LIN {X 0,Y 462.076,Z 805.62,A -85,B 0,C 180,E1 21191.71,E2 21191.71} C_VEL
LIN {X 0,Y 459.334,Z 826.839,A -85,B 0,C 180,E1 21190.527,E2 21190.527} C_VEL
LIN {X 0,Y 456.263,Z 847.373,A -85,B 0,C 180,E1 21189.127,E2 21189.127} C_VEL
LIN {X 0,Y 453.108,Z 867.434,A -85,B 0,C 180,E1 21187.515,E2 21187.515} C_VEL
LIN {X 0,Y 449.988,Z 885.995,A -85,B 0,C 180,E1 21185.755,E2 21185.755} C_VEL
LIN {X 0,Y 446.558,Z 905.771,A -85,B 0,C 180,E1 21183.572,E2 21183.572} C_VEL
LIN {X 0,Y 443.731,Z 922.212,A -85,B 0,C 180,E1 21181.463,E2 21181.463} C_VEL
LIN {X 0,Y 440.914,Z 938.619,A -85,B 0,C 180,E1 21179.028,E2 21179.028} C_VEL
LIN {X 0,Y 438.594,Z 953.242,A -85,B 0,C 180,E1 21176.537,E2 21176.537} C_VEL
LIN {X 0,Y 436.587,Z 966.429,A -85,B 0,C 180,E1 21173.911,E2 21173.911} C_VEL
LIN {X 0,Y 434.952,Z 978.265,A -85,B 0,C 180,E1 21171.154,E2 21171.154} C_VEL
LIN {X 0,Y 433.708,Z 988.605,A -85,B 0,C 180,E1 21168.27,E2 21168.27} C_VEL
LIN {X 0,Y 432.814,Z 997.995,A -85,B 0,C 180,E1 21165.131,E2 21165.131} C_VEL
LIN {X 0,Y 432.337,Z 1004.562,A -85,B 0,C 180,E1 21162.419,E2 21162.419} C_VEL
LIN {X 0,Y 432.051,Z 1010.43,A -85,B 0,C 180,E1 21159.322,E2 21159.322} C_VEL
LIN {X 0,Y 431.943,Z 1014.119,A -85,B 0,C 180,E1 21156.646,E2 21156.646} C_VEL
LIN {X 0,Y 431.896,Z 1016.848,A -85,B 0,C 180,E1 21153.584,E2 21153.584} C_VEL
LIN {X 0,Y 431.89,Z 1017.848,A -85,B 0,C 180,E1 21150.929,E2 21150.929} C_VEL
LIN {X 0,Y 431.907,Z 1017.69,A -85,B 0,C 180,E1 21148.143,E2 21148.143} C_VEL
LIN {X 0,Y 431.91,Z 1015.955,A -85,B 0,C 180,E1 21145.22,E2 21145.22} C_VEL
LIN {X 0,Y 431.948,Z 1013.161,A -85,B 0,C 180,E1 21142.553,E2 21142.553} C_VEL
LIN {X 0,Y 432.128,Z 1008.339,A -85,B 0,C 180,E1 21139.469,E2 21139.469} C_VEL
LIN {X 0,Y 432.462,Z 1002.684,A -85,B 0,C 180,E1 21136.743,E2 21136.743} C_VEL
LIN {X 0,Y 433.106,Z 994.557,A -85,B 0,C 180,E1 21133.644,E2 21133.644} C_VEL
LIN {X 0,Y 434.06,Z 985.527,A -85,B 0,C 180,E1 21130.809,E2 21130.809} C_VEL
LIN {X 0,Y 435.394,Z 974.873,A -85,B 0,C 180,E1 21128.021,E2 21128.021} C_VEL
LIN {X 0,Y 436.966,Z 963.844,A -85,B 0,C 180,E1 21125.537,E2 21125.537} C_VEL
LIN {X 0,Y 439.061,Z 950.109,A -85,B 0,C 180,E1 21122.91,E2 21122.91} C_VEL
LIN {X 0,Y 441.553,Z 935.071,A -85,B 0,C 180,E1 21120.404,E2 21120.404} C_VEL
LIN {X 0,Y 444.365,Z 918.393,A -85,B 0,C 180,E1 21118.024,E2 21118.024} C_VEL
LIN {X 0,Y 447.495,Z 900.571,A -85,B 0,C 180,E1 21115.815,E2 21115.815} C_VEL
LIN {X 0,Y 450.434,Z 883.294,A -85,B 0,C 180,E1 21113.973,E2 21113.973} C_VEL
LIN {X 0,Y 453.737,Z 863.496,A -85,B 0,C 180,E1 21112.148,E2 21112.148} C_VEL
LIN {X 0,Y 456.694,Z 844.645,A -85,B 0,C 180,E1 21110.674,E2 21110.674} C_VEL
LIN {X 0,Y 459.9,Z 822.472,A -85,B 0,C 180,E1 21109.215,E2 21109.215} C_VEL
LIN {X 0,Y 462.377,Z 803.115,A -85,B 0,C 180,E1 21108.162,E2 21108.162} C_VEL
LIN {X 0,Y 465.009,Z 779.05,A -85,B 0,C 180,E1 21107.112,E2 21107.112} C_VEL
LIN {X 0,Y 467.004,Z 756.997,A -85,B 0,C 180,E1 21106.38,E2 21106.38} C_VEL
LIN {X 0,Y 468.458,Z 733.73,A -85,B 0,C 180,E1 21105.834,E2 21105.834} C_VEL
LIN {X 0,Y 474.656,Z 531.518,A -85,B 0,C 180,E1 21102.256,E2 21102.256} C_VEL
LIN {X 0,Y 477.415,Z 442.989,A -85,B 0,C 180,E1 21100.663,E2 21100.663} C_VEL
LIN {X 0,Y 466.316,Z 425.345,A -85,B 0,C 180,E1 21098.644,E2 21098.644} C_VEL
LIN {X 0,Y 456.213,Z 410.687,A -85,B 0,C 180,E1 21096.671,E2 21096.671} C_VEL
LIN {X 0,Y 446.549,Z 397.276,A -85,B 0,C 180,E1 21094.622,E2 21094.622} C_VEL
LIN {X 0,Y 442.193,Z 391.483,A -85,B 0,C 180,E1 21093.64,E2 21093.64} C_VEL
LIN {X 0,Y 438.295,Z 386.486,A -85,B 0,C 180,E1 21092.728,E2 21092.728} C_VEL
LIN {X 0,Y 436.603,Z 384.125,A -85,B 0,C 180,E1 21092.248,E2 21092.248} C_VEL
LIN {X 0,Y 435.545,Z 381.762,A -85,B 0,C 180,E1 21091.715,E2 21091.715} C_VEL
LIN {X 0,Y 433.675,Z 378.949,A -85,B 0,C 180,E1 21090.939,E2 21090.939} C_VEL
LIN {X 0,Y 433.213,Z 377.052,A -85,B 0,C 180,E1 21090.514,E2 21090.514} C_VEL
LIN {X 0,Y 433.202,Z 377.083,A -85,B 0,C 180,E1 21086.748,E2 21086.748} C_VEL
LIN {X 0,Y 433.196,Z 377.04,A -85,B 0,C 180,E1 21082.954,E2 21082.954} C_VEL
LIN {X 0,Y 433.235,Z 377.058,A -85,B 0,C 180,E1 21079.41,E2 21079.41} C_VEL
LIN {X 0,Y 433.241,Z 377.062,A -85,B 0,C 180,E1 21075.528,E2 21075.528} C_VEL
LIN {X 0,Y 433.199,Z 377.077,A -85,B 0,C 180,E1 21071.854,E2 21071.854} C_VEL
LIN {X 0,Y 433.177,Z 377.084,A -85,B 0,C 180,E1 21068.227,E2 21068.227} C_VEL
LIN {X 0,Y 433.183,Z 377.087,A -85,B 0,C 180,E1 21064.434,E2 21064.434} C_VEL
LIN {X 0,Y 433.218,Z 377.081,A -85,B 0,C 180,E1 21060.793,E2 21060.793} C_VEL
LIN {X 0,Y 433.232,Z 377.079,A -85,B 0,C 180,E1 21057.089,E2 21057.089} C_VEL
LIN {X 0,Y 433.208,Z 377.083,A -85,B 0,C 180,E1 21053.373,E2 21053.373} C_VEL
LIN {X 0,Y 433.195,Z 377.086,A -85,B 0,C 180,E1 21049.763,E2 21049.763} C_VEL
LIN {X 0,Y 433.206,Z 377.086,A -85,B 0,C 180,E1 21045.975,E2 21045.975} C_VEL
LIN {X 0,Y 433.24,Z 377.03,A -85,B 0,C 180,E1 21042.37,E2 21042.37} C_VEL
LIN {X 0,Y 433.253,Z 377.074,A -85,B 0,C 180,E1 21038.615,E2 21038.615} C_VEL
LIN {X 0,Y 433.225,Z 377.048,A -85,B 0,C 180,E1 21034.871,E2 21034.871} C_VEL
LIN {X 0,Y 433.213,Z 377.045,A -85,B 0,C 180,E1 21031.159,E2 21031.159} C_VEL
LIN {X 0,Y 433.277,Z 377.224,A -85,B 0,C 180,E1 21028.021,E2 21028.021} C_VEL
LIN {X 0,Y 434.29,Z 380.161,A -85,B 0,C 180,E1 21027.715,E2 21027.715} C_VEL
LIN {X 0,Y 436.695,Z 382.725,A -85,B 0,C 180,E1 21027.137,E2 21027.137} C_VEL
LIN {X 0,Y 438.075,Z 383.765,A -85,B 0,C 180,E1 21026.824,E2 21026.824} C_VEL
LIN {X 0,Y 440.43,Z 387.482,A -85,B 0,C 180,E1 21026.246,E2 21026.246} C_VEL
LIN {X 0,Y 442.869,Z 389.914,A -85,B 0,C 180,E1 21025.702,E2 21025.702} C_VEL
LIN {X 0,Y 446.063,Z 394.129,A -85,B 0,C 180,E1 21024.982,E2 21024.982} C_VEL
LIN {X 0,Y 447.593,Z 395.982,A -85,B 0,C 180,E1 21024.65,E2 21024.65} C_VEL
LIN {X 0,Y 456.054,Z 406.862,A -85,B 0,C 180,E1 21022.882,E2 21022.882} C_VEL
LIN {X 0,Y 467.056,Z 421.727,A -85,B 0,C 180,E1 21020.758,E2 21020.758} C_VEL
LIN {X 0,Y 477.318,Z 436.615,A -85,B 0,C 180,E1 21018.921,E2 21018.921} C_VEL
LIN {X 0,Y 470.969,Z 637.153,A -85,B 0,C 180,E1 21015.357,E2 21015.357} C_VEL
LIN {X 0,Y 469.061,Z 701.067,A -85,B 0,C 180,E1 21014.235,E2 21014.235} C_VEL
LIN {X 0,Y 467.994,Z 708.752,A -85,B 0,C 180,E1 21014.173,E2 21014.173} C_VEL
LIN {X 0,Y 462.507,Z 728.147,A -85,B 0,C 180,E1 21014.247,E2 21014.247} C_VEL
LIN {X 0,Y 461.232,Z 735.659,A -85,B 0,C 180,E1 21014.106,E2 21014.106} C_VEL
LIN {X 0,Y 459.247,Z 757.338,A -85,B 0,C 180,E1 21013.336,E2 21013.336} C_VEL
LIN {X 0,Y 456.812,Z 778.149,A -85,B 0,C 180,E1 21012.381,E2 21012.381} C_VEL
LIN {X 0,Y 454.246,Z 797.149,A -85,B 0,C 180,E1 21011.32,E2 21011.32} C_VEL
LIN {X 0,Y 450.876,Z 818.833,A -85,B 0,C 180,E1 21009.852,E2 21009.852} C_VEL
LIN {X 0,Y 447.624,Z 838.068,A -85,B 0,C 180,E1 21008.3,E2 21008.3} C_VEL
LIN {X 0,Y 444.229,Z 856.539,A -85,B 0,C 180,E1 21006.532,E2 21006.532} C_VEL
LIN {X 0,Y 440.833,Z 874.551,A -85,B 0,C 180,E1 21004.538,E2 21004.538} C_VEL
LIN {X 0,Y 437.468,Z 891.506,A -85,B 0,C 180,E1 21002.327,E2 21002.327} C_VEL
LIN {X 0,Y 434.438,Z 907.273,A -85,B 0,C 180,E1 20999.958,E2 20999.958} C_VEL
LIN {X 0,Y 431.785,Z 921.227,A -85,B 0,C 180,E1 20997.515,E2 20997.515} C_VEL
LIN {X 0,Y 429.286,Z 935.376,A -85,B 0,C 180,E1 20994.636,E2 20994.636} C_VEL
LIN {X 0,Y 427.507,Z 946.566,A -85,B 0,C 180,E1 20991.972,E2 20991.972} C_VEL
LIN {X 0,Y 425.948,Z 958.005,A -85,B 0,C 180,E1 20988.756,E2 20988.756} C_VEL
LIN {X 0,Y 425.016,Z 966.889,A -85,B 0,C 180,E1 20985.807,E2 20985.807} C_VEL
LIN {X 0,Y 424.426,Z 973.858,A -85,B 0,C 180,E1 20982.93,E2 20982.93} C_VEL
LIN {X 0,Y 424.076,Z 979.744,A -85,B 0,C 180,E1 20979.909,E2 20979.909} C_VEL
LIN {X 0,Y 423.936,Z 983.747,A -85,B 0,C 180,E1 20977.043,E2 20977.043} C_VEL
LIN {X 0,Y 423.913,Z 986.485,A -85,B 0,C 180,E1 20974.192,E2 20974.192} C_VEL
LIN {X 0,Y 423.905,Z 987.795,A -85,B 0,C 180,E1 20971.216,E2 20971.216} C_VEL
LIN {X 0,Y 423.909,Z 987.765,A -85,B 0,C 180,E1 20968.513,E2 20968.513} C_VEL
LIN {X 0,Y 423.907,Z 986.22,A -85,B 0,C 180,E1 20965.4,E2 20965.4} C_VEL
LIN {X 0,Y 423.934,Z 983.693,A -85,B 0,C 180,E1 20962.82,E2 20962.82} C_VEL
LIN {X 0,Y 424.08,Z 979.671,A -85,B 0,C 180,E1 20959.953,E2 20959.953} C_VEL
LIN {X 0,Y 424.438,Z 973.751,A -85,B 0,C 180,E1 20956.931,E2 20956.931} C_VEL
LIN {X 0,Y 425.066,Z 966.304,A -85,B 0,C 180,E1 20953.887,E2 20953.887} C_VEL
LIN {X 0,Y 426.021,Z 957.373,A -85,B 0,C 180,E1 20950.962,E2 20950.962} C_VEL
LIN {X 0,Y 427.696,Z 945.224,A -85,B 0,C 180,E1 20947.603,E2 20947.603} C_VEL
LIN {X 0,Y 429.668,Z 933.263,A -85,B 0,C 180,E1 20944.798,E2 20944.798} C_VEL
LIN {X 0,Y 432.036,Z 919.809,A -85,B 0,C 180,E1 20942.132,E2 20942.132} C_VEL
LIN {X 0,Y 434.919,Z 904.789,A -85,B 0,C 180,E1 20939.554,E2 20939.554} C_VEL
LIN {X 0,Y 437.948,Z 889.086,A -85,B 0,C 180,E1 20937.246,E2 20937.246} C_VEL
LIN {X 0,Y 441.59,Z 870.435,A -85,B 0,C 180,E1 20934.897,E2 20934.897} C_VEL
LIN {X 0,Y 444.969,Z 852.67,A -85,B 0,C 180,E1 20932.977,E2 20932.977} C_VEL
LIN {X 0,Y 448.437,Z 833.332,A -85,B 0,C 180,E1 20931.21,E2 20931.21} C_VEL
LIN {X 0,Y 451.792,Z 813.522,A -85,B 0,C 180,E1 20929.665,E2 20929.665} C_VEL
LIN {X 0,Y 454.832,Z 792.848,A -85,B 0,C 180,E1 20928.333,E2 20928.333} C_VEL
LIN {X 0,Y 457.698,Z 770.919,A -85,B 0,C 180,E1 20927.167,E2 20927.167} C_VEL
LIN {X 0,Y 459.99,Z 749.57,A -85,B 0,C 180,E1 20926.274,E2 20926.274} C_VEL
LIN {X 0,Y 462.016,Z 725.777,A -85,B 0,C 180,E1 20925.523,E2 20925.523} C_VEL
LIN {X 0,Y 463.236,Z 704.237,A -85,B 0,C 180,E1 20925.041,E2 20925.041} C_VEL
LIN {X 0,Y 470.098,Z 495.365,A -85,B 0,C 180,E1 20921.31,E2 20921.31} C_VEL
LIN {X 0,Y 471.926,Z 440.345,A -85,B 0,C 180,E1 20920.306,E2 20920.306} C_VEL
LIN {X 0,Y 460.786,Z 424.412,A -85,B 0,C 180,E1 20918.237,E2 20918.237} C_VEL
LIN {X 0,Y 451.359,Z 411.585,A -85,B 0,C 180,E1 20916.34,E2 20916.34} C_VEL
LIN {X 0,Y 446.19,Z 405.119,A -85,B 0,C 180,E1 20915.242,E2 20915.242} C_VEL
LIN {X 0,Y 442.926,Z 400.842,A -85,B 0,C 180,E1 20914.514,E2 20914.514} C_VEL
LIN {X 0,Y 438.862,Z 395.672,A -85,B 0,C 180,E1 20913.577,E2 20913.577} C_VEL
LIN {X 0,Y 435.602,Z 391.675,A -85,B 0,C 180,E1 20912.8,E2 20912.8} C_VEL
LIN {X 0,Y 434.669,Z 390.322,A -85,B 0,C 180,E1 20912.566,E2 20912.566} C_VEL
LIN {X 0,Y 431.553,Z 387.217,A -85,B 0,C 180,E1 20911.809,E2 20911.809} C_VEL
LIN {X 0,Y 430.027,Z 384.394,A -85,B 0,C 180,E1 20911.388,E2 20911.388} C_VEL
LIN {X 0,Y 427.064,Z 382.162,A -85,B 0,C 180,E1 20910.651,E2 20910.651} C_VEL
LIN {X 0,Y 425.547,Z 379.242,A -85,B 0,C 180,E1 20910.205,E2 20910.205} C_VEL
LIN {X 0,Y 425.308,Z 378.027,A -85,B 0,C 180,E1 20910.092,E2 20910.092} C_VEL
LIN {X 0,Y 425.286,Z 378.074,A -85,B 0,C 180,E1 20906.382,E2 20906.382} C_VEL
LIN {X 0,Y 425.271,Z 378.03,A -85,B 0,C 180,E1 20902.499,E2 20902.499} C_VEL
LIN {X 0,Y 425.271,Z 378.039,A -85,B 0,C 180,E1 20898.648,E2 20898.648} C_VEL
LIN {X 0,Y 425.29,Z 378.051,A -85,B 0,C 180,E1 20894.949,E2 20894.949} C_VEL
LIN {X 0,Y 425.31,Z 378.059,A -85,B 0,C 180,E1 20891.252,E2 20891.252} C_VEL
LIN {X 0,Y 425.291,Z 378.064,A -85,B 0,C 180,E1 20887.43,E2 20887.43} C_VEL
LIN {X 0,Y 425.257,Z 378.07,A -85,B 0,C 180,E1 20883.775,E2 20883.775} C_VEL
LIN {X 0,Y 425.25,Z 378.073,A -85,B 0,C 180,E1 20880,E2 20880} C_VEL
LIN {X 0,Y 425.254,Z 378.074,A -85,B 0,C 180,E1 20876.226,E2 20876.226} C_VEL
LIN {X 0,Y 425.285,Z 378.07,A -85,B 0,C 180,E1 20872.571,E2 20872.571} C_VEL
LIN {X 0,Y 425.289,Z 378.074,A -85,B 0,C 180,E1 20868.748,E2 20868.748} C_VEL
LIN {X 0,Y 425.263,Z 378.075,A -85,B 0,C 180,E1 20865.012,E2 20865.012} C_VEL
LIN {X 0,Y 425.247,Z 378.035,A -85,B 0,C 180,E1 20861.342,E2 20861.342} C_VEL
LIN {X 0,Y 425.254,Z 378.044,A -85,B 0,C 180,E1 20857.506,E2 20857.506} C_VEL
LIN {X 0,Y 425.279,Z 378.073,A -85,B 0,C 180,E1 20853.769,E2 20853.769} C_VEL
LIN {X 0,Y 425.291,Z 378.258,A -85,B 0,C 180,E1 20851.033,E2 20851.033} C_VEL
LIN {X 0,Y 426.687,Z 381.61,A -85,B 0,C 180,E1 20850.213,E2 20850.213} C_VEL
LIN {X 0,Y 428.223,Z 383.778,A -85,B 0,C 180,E1 20849.558,E2 20849.558} C_VEL
LIN {X 0,Y 431.134,Z 387.942,A -85,B 0,C 180,E1 20848.742,E2 20848.742} C_VEL
LIN {X 0,Y 432.999,Z 390.22,A -85,B 0,C 180,E1 20848.271,E2 20848.271} C_VEL
LIN {X 0,Y 440.536,Z 400.021,A -85,B 0,C 180,E1 20846.451,E2 20846.451} C_VEL
LIN {X 0,Y 451.037,Z 414.496,A -85,B 0,C 180,E1 20844.122,E2 20844.122} C_VEL
LIN {X 0,Y 462.686,Z 431.668,A -85,B 0,C 180,E1 20841.768,E2 20841.768} C_VEL
LIN {X 0,Y 472.168,Z 446.874,A -85,B 0,C 180,E1 20839.991,E2 20839.991} C_VEL
LIN {X 0,Y 465.285,Z 654.823,A -85,B 0,C 180,E1 20836.266,E2 20836.266} C_VEL
LIN {X 0,Y 462.484,Z 738.649,A -85,B 0,C 180,E1 20834.757,E2 20834.757} C_VEL
LIN {X 0,Y 460.69,Z 762.093,A -85,B 0,C 180,E1 20834.15,E2 20834.15} C_VEL
LIN {X 0,Y 458.499,Z 784.883,A -85,B 0,C 180,E1 20833.339,E2 20833.339} C_VEL
LIN {X 0,Y 455.988,Z 805.515,A -85,B 0,C 180,E1 20832.383,E2 20832.383} C_VEL
LIN {X 0,Y 453.13,Z 826.558,A -85,B 0,C 180,E1 20831.199,E2 20831.199} C_VEL
LIN {X 0,Y 449.902,Z 847.049,A -85,B 0,C 180,E1 20829.79,E2 20829.79} C_VEL
LIN {X 0,Y 446.417,Z 867.865,A -85,B 0,C 180,E1 20828.096,E2 20828.096} C_VEL
LIN {X 0,Y 443.189,Z 886.014,A -85,B 0,C 180,E1 20826.351,E2 20826.351} C_VEL
LIN {X 0,Y 439.612,Z 905.458,A -85,B 0,C 180,E1 20824.175,E2 20824.175} C_VEL
LIN {X 0,Y 436.562,Z 922.064,A -85,B 0,C 180,E1 20822.016,E2 20822.016} C_VEL
LIN {X 0,Y 433.595,Z 938.304,A -85,B 0,C 180,E1 20819.566,E2 20819.566} C_VEL
LIN {X 0,Y 431.107,Z 952.927,A -85,B 0,C 180,E1 20817.035,E2 20817.035} C_VEL
LIN {X 0,Y 428.887,Z 966.491,A -85,B 0,C 180,E1 20814.283,E2 20814.283} C_VEL
LIN {X 0,Y 427.137,Z 978.706,A -85,B 0,C 180,E1 20811.416,E2 20811.416} C_VEL
LIN {X 0,Y 425.929,Z 988.145,A -85,B 0,C 180,E1 20808.758,E2 20808.758} C_VEL
LIN {X 0,Y 424.975,Z 997.288,A -85,B 0,C 180,E1 20805.696,E2 20805.696} C_VEL
LIN {X 0,Y 424.4,Z 1004.259,A -85,B 0,C 180,E1 20802.794,E2 20802.794} C_VEL
LIN {X 0,Y 424.064,Z 1010.224,A -85,B 0,C 180,E1 20799.636,E2 20799.636} C_VEL
LIN {X 0,Y 423.937,Z 1013.959,A -85,B 0,C 180,E1 20796.908,E2 20796.908} C_VEL
LIN {X 0,Y 423.909,Z 1016.732,A -85,B 0,C 180,E1 20793.881,E2 20793.881} C_VEL
LIN {X 0,Y 423.896,Z 1017.826,A -85,B 0,C 180,E1 20791.081,E2 20791.081} C_VEL
LIN {X 0,Y 423.906,Z 1017.735,A -85,B 0,C 180,E1 20788.379,E2 20788.379} C_VEL
LIN {X 0,Y 423.909,Z 1016.068,A -85,B 0,C 180,E1 20785.266,E2 20785.266} C_VEL
LIN {X 0,Y 423.95,Z 1013.321,A -85,B 0,C 180,E1 20782.548,E2 20782.548} C_VEL
LIN {X 0,Y 424.142,Z 1008.593,A -85,B 0,C 180,E1 20779.406,E2 20779.406} C_VEL
LIN {X 0,Y 424.498,Z 1002.921,A -85,B 0,C 180,E1 20776.598,E2 20776.598} C_VEL
LIN {X 0,Y 425.181,Z 994.96,A -85,B 0,C 180,E1 20773.471,E2 20773.471} C_VEL
LIN {X 0,Y 426.153,Z 986.316,A -85,B 0,C 180,E1 20770.684,E2 20770.684} C_VEL
LIN {X 0,Y 427.6,Z 975.301,A -85,B 0,C 180,E1 20767.743,E2 20767.743} C_VEL
LIN {X 0,Y 429.36,Z 963.53,A -85,B 0,C 180,E1 20765.074,E2 20765.074} C_VEL
LIN {X 0,Y 431.596,Z 949.794,A -85,B 0,C 180,E1 20762.402,E2 20762.402} C_VEL
LIN {X 0,Y 434.254,Z 934.872,A -85,B 0,C 180,E1 20759.876,E2 20759.876} C_VEL
LIN {X 0,Y 437.203,Z 918.471,A -85,B 0,C 180,E1 20757.496,E2 20757.496} C_VEL
LIN {X 0,Y 440.5,Z 900.874,A -85,B 0,C 180,E1 20755.274,E2 20755.274} C_VEL
LIN {X 0,Y 443.719,Z 882.978,A -85,B 0,C 180,E1 20753.34,E2 20753.34} C_VEL
LIN {X 0,Y 447.368,Z 862.366,A -85,B 0,C 180,E1 20751.429,E2 20751.429} C_VEL
LIN {X 0,Y 450.415,Z 843.96,A -85,B 0,C 180,E1 20749.982,E2 20749.982} C_VEL
LIN {X 0,Y 453.761,Z 821.849,A -85,B 0,C 180,E1 20748.519,E2 20748.519} C_VEL
LIN {X 0,Y 456.492,Z 801.511,A -85,B 0,C 180,E1 20747.412,E2 20747.412} C_VEL
LIN {X 0,Y 459.155,Z 778.271,A -85,B 0,C 180,E1 20746.407,E2 20746.407} C_VEL
LIN {X 0,Y 461.272,Z 755.966,A -85,B 0,C 180,E1 20745.668,E2 20745.668} C_VEL
LIN {X 0,Y 462.752,Z 732.697,A -85,B 0,C 180,E1 20745.126,E2 20745.126} C_VEL
LIN {X 0,Y 469.367,Z 528.448,A -85,B 0,C 180,E1 20741.479,E2 20741.479} C_VEL
LIN {X 0,Y 472.023,Z 446.625,A -85,B 0,C 180,E1 20739.987,E2 20739.987} C_VEL
LIN {X 0,Y 461.095,Z 429.391,A -85,B 0,C 180,E1 20737.934,E2 20737.934} C_VEL
LIN {X 0,Y 450.293,Z 413.43,A -85,B 0,C 180,E1 20735.731,E2 20735.731} C_VEL
LIN {X 0,Y 442.69,Z 403.108,A -85,B 0,C 180,E1 20734.064,E2 20734.064} C_VEL
LIN {X 0,Y 438.897,Z 397.933,A -85,B 0,C 180,E1 20733.183,E2 20733.183} C_VEL
LIN {X 0,Y 431.55,Z 388.337,A -85,B 0,C 180,E1 20731.38,E2 20731.38} C_VEL
LIN {X 0,Y 428.463,Z 384.385,A -85,B 0,C 180,E1 20730.578,E2 20730.578} C_VEL
LIN {X 0,Y 427.616,Z 382.741,A -85,B 0,C 180,E1 20730.179,E2 20730.179} C_VEL
LIN {X 0,Y 425.603,Z 379.511,A -85,B 0,C 180,E1 20729.251,E2 20729.251} C_VEL
LIN {X 0,Y 425.261,Z 378.027,A -85,B 0,C 180,E1 20728.912,E2 20728.912} C_VEL
LIN {X 0,Y 425.271,Z 378.038,A -85,B 0,C 180,E1 20725.168,E2 20725.168} C_VEL
LIN {X 0,Y 425.298,Z 378.057,A -85,B 0,C 180,E1 20721.43,E2 20721.43} C_VEL
LIN {X 0,Y 425.292,Z 378.017,A -85,B 0,C 180,E1 20717.654,E2 20717.654} C_VEL
LIN {X 0,Y 425.259,Z 378.077,A -85,B 0,C 180,E1 20714.014,E2 20714.014} C_VEL
LIN {X 0,Y 425.242,Z 378.077,A -85,B 0,C 180,E1 20710.293,E2 20710.293} C_VEL
LIN {X 0,Y 425.242,Z 378.072,A -85,B 0,C 180,E1 20706.48,E2 20706.48} C_VEL
LIN {X 0,Y 425.273,Z 378.065,A -85,B 0,C 180,E1 20702.83,E2 20702.83} C_VEL
LIN {X 0,Y 425.303,Z 378.06,A -85,B 0,C 180,E1 20699.057,E2 20699.057} C_VEL
LIN {X 0,Y 425.286,Z 378.061,A -85,B 0,C 180,E1 20695.145,E2 20695.145} C_VEL
LIN {X 0,Y 425.256,Z 378.066,A -85,B 0,C 180,E1 20691.618,E2 20691.618} C_VEL
LIN {X 0,Y 425.259,Z 378.062,A -85,B 0,C 180,E1 20687.783,E2 20687.783} C_VEL
LIN {X 0,Y 425.273,Z 378.038,A -85,B 0,C 180,E1 20684.033,E2 20684.033} C_VEL
LIN {X 0,Y 425.308,Z 378.052,A -85,B 0,C 180,E1 20680.355,E2 20680.355} C_VEL
LIN {X 0,Y 425.308,Z 378.02,A -85,B 0,C 180,E1 20676.59,E2 20676.59} C_VEL
LIN {X 0,Y 425.298,Z 378.066,A -85,B 0,C 180,E1 20672.713,E2 20672.713} C_VEL
LIN {X 0,Y 425.322,Z 378.231,A -85,B 0,C 180,E1 20669.768,E2 20669.768} C_VEL
LIN {X 0,Y 426.31,Z 381.08,A -85,B 0,C 180,E1 20669.445,E2 20669.445} C_VEL
LIN {X 0,Y 428.708,Z 383.661,A -85,B 0,C 180,E1 20668.818,E2 20668.818} C_VEL
LIN {X 0,Y 430.265,Z 384.812,A -85,B 0,C 180,E1 20668.436,E2 20668.436} C_VEL
LIN {X 0,Y 432.502,Z 388.462,A -85,B 0,C 180,E1 20667.839,E2 20667.839} C_VEL
LIN {X 0,Y 435.233,Z 391.028,A -85,B 0,C 180,E1 20667.188,E2 20667.188} C_VEL
LIN {X 0,Y 438.272,Z 395.141,A -85,B 0,C 180,E1 20666.45,E2 20666.45} C_VEL
LIN {X 0,Y 440.005,Z 397.069,A -85,B 0,C 180,E1 20666.052,E2 20666.052} C_VEL
LIN {X 0,Y 443.745,Z 401.631,A -85,B 0,C 180,E1 20665.206,E2 20665.206} C_VEL
LIN {X 0,Y 447.929,Z 407.057,A -85,B 0,C 180,E1 20664.287,E2 20664.287} C_VEL
LIN {X 0,Y 459.725,Z 422.893,A -85,B 0,C 180,E1 20661.873,E2 20661.873} C_VEL
LIN {X 0,Y 471.903,Z 440.34,A -85,B 0,C 180,E1 20659.603,E2 20659.603} C_VEL
LIN {X 0,Y 466.158,Z 613.48,A -85,B 0,C 180,E1 20656.484,E2 20656.484} C_VEL
LIN {X 0,Y 462.793,Z 713.541,A -85,B 0,C 180,E1 20654.685,E2 20654.685} C_VEL
LIN {X 0,Y 461.232,Z 735.659,A -85,B 0,C 180,E1 20654.106,E2 20654.106} C_VEL
LIN {X 0,Y 460.05,Z 742.122,A -85,B 0,C 180,E1 20653.984,E2 20653.984} C_VEL
LIN {X 0,Y 453.544,Z 762.396,A -85,B 0,C 180,E1 20653.752,E2 20653.752} C_VEL
LIN {X 0,Y 452.005,Z 769.58,A -85,B 0,C 180,E1 20653.511,E2 20653.511} C_VEL
LIN {X 0,Y 448.953,Z 792.198,A -85,B 0,C 180,E1 20652.32,E2 20652.32} C_VEL
LIN {X 0,Y 445.931,Z 811.777,A -85,B 0,C 180,E1 20651.062,E2 20651.062} C_VEL
LIN {X 0,Y 442.416,Z 831.963,A -85,B 0,C 180,E1 20649.502,E2 20649.502} C_VEL
LIN {X 0,Y 438.882,Z 850.841,A -85,B 0,C 180,E1 20647.789,E2 20647.789} C_VEL
LIN {X 0,Y 435.147,Z 869.369,A -85,B 0,C 180,E1 20645.796,E2 20645.796} C_VEL
LIN {X 0,Y 431.598,Z 886.832,A -85,B 0,C 180,E1 20643.615,E2 20643.615} C_VEL
LIN {X 0,Y 428.272,Z 902.658,A -85,B 0,C 180,E1 20641.298,E2 20641.298} C_VEL
LIN {X 0,Y 424.977,Z 918.917,A -85,B 0,C 180,E1 20638.525,E2 20638.525} C_VEL
LIN {X 0,Y 422.474,Z 931.977,A -85,B 0,C 180,E1 20635.929,E2 20635.929} C_VEL
LIN {X 0,Y 420.299,Z 944.075,A -85,B 0,C 180,E1 20633.108,E2 20633.108} C_VEL
LIN {X 0,Y 418.632,Z 954.868,A -85,B 0,C 180,E1 20630.175,E2 20630.175} C_VEL
LIN {X 0,Y 417.399,Z 964.085,A -85,B 0,C 180,E1 20627.134,E2 20627.134} C_VEL
LIN {X 0,Y 416.572,Z 972.648,A -85,B 0,C 180,E1 20623.744,E2 20623.744} C_VEL
LIN {X 0,Y 416.188,Z 978.257,A -85,B 0,C 180,E1 20620.939,E2 20620.939} C_VEL
LIN {X 0,Y 415.977,Z 983.109,A -85,B 0,C 180,E1 20617.734,E2 20617.734} C_VEL
LIN {X 0,Y 415.917,Z 985.917,A -85,B 0,C 180,E1 20614.964,E2 20614.964} C_VEL
LIN {X 0,Y 415.907,Z 987.682,A -85,B 0,C 180,E1 20611.928,E2 20611.928} C_VEL
LIN {X 0,Y 415.888,Z 987.855,A -85,B 0,C 180,E1 20609.035,E2 20609.035} C_VEL
LIN {X 0,Y 415.9,Z 986.87,A -85,B 0,C 180,E1 20606.278,E2 20606.278} C_VEL
LIN {X 0,Y 415.938,Z 984.171,A -85,B 0,C 180,E1 20603.097,E2 20603.097} C_VEL
LIN {X 0,Y 416.063,Z 980.703,A -85,B 0,C 180,E1 20600.456,E2 20600.456} C_VEL
LIN {X 0,Y 416.403,Z 974.961,A -85,B 0,C 180,E1 20597.239,E2 20597.239} C_VEL
LIN {X 0,Y 416.953,Z 968.458,A -85,B 0,C 180,E1 20594.422,E2 20594.422} C_VEL
LIN {X 0,Y 418.057,Z 958.933,A -85,B 0,C 180,E1 20591.02,E2 20591.02} C_VEL
LIN {X 0,Y 419.46,Z 949.345,A -85,B 0,C 180,E1 20588.172,E2 20588.172} C_VEL
LIN {X 0,Y 421.375,Z 937.925,A -85,B 0,C 180,E1 20585.318,E2 20585.318} C_VEL
LIN {X 0,Y 423.874,Z 924.774,A -85,B 0,C 180,E1 20582.49,E2 20582.49} C_VEL
LIN {X 0,Y 426.74,Z 910.151,A -85,B 0,C 180,E1 20579.834,E2 20579.834} C_VEL
LIN {X 0,Y 430.2,Z 893.383,A -85,B 0,C 180,E1 20577.216,E2 20577.216} C_VEL
LIN {X 0,Y 433.586,Z 877.133,A -85,B 0,C 180,E1 20575.041,E2 20575.041} C_VEL
LIN {X 0,Y 437.304,Z 858.731,A -85,B 0,C 180,E1 20572.936,E2 20572.936} C_VEL
LIN {X 0,Y 440.96,Z 840.01,A -85,B 0,C 180,E1 20571.096,E2 20571.096} C_VEL
LIN {X 0,Y 444.505,Z 820.092,A -85,B 0,C 180,E1 20569.458,E2 20569.458} C_VEL
LIN {X 0,Y 447.961,Z 799.179,A -85,B 0,C 180,E1 20568.01,E2 20568.01} C_VEL
LIN {X 0,Y 450.714,Z 779.792,A -85,B 0,C 180,E1 20566.907,E2 20566.907} C_VEL
LIN {X 0,Y 453.382,Z 758.272,A -85,B 0,C 180,E1 20565.9,E2 20565.9} C_VEL
LIN {X 0,Y 455.498,Z 736.206,A -85,B 0,C 180,E1 20565.109,E2 20565.109} C_VEL
LIN {X 0,Y 457.225,Z 712.305,A -85,B 0,C 180,E1 20564.488,E2 20564.488} C_VEL
LIN {X 0,Y 463.98,Z 519.972,A -85,B 0,C 180,E1 20561.01,E2 20561.01} C_VEL
LIN {X 0,Y 466.634,Z 444.332,A -85,B 0,C 180,E1 20559.622,E2 20559.622} C_VEL
LIN {X 0,Y 455.006,Z 427.591,A -85,B 0,C 180,E1 20557.377,E2 20557.377} C_VEL
LIN {X 0,Y 444.492,Z 413.468,A -85,B 0,C 180,E1 20555.16,E2 20555.16} C_VEL
LIN {X 0,Y 439.236,Z 406.899,A -85,B 0,C 180,E1 20553.976,E2 20553.976} C_VEL
LIN {X 0,Y 435.595,Z 402.233,A -85,B 0,C 180,E1 20553.114,E2 20553.114} C_VEL
LIN {X 0,Y 431.57,Z 397.15,A -85,B 0,C 180,E1 20552.121,E2 20552.121} C_VEL
LIN {X 0,Y 428.304,Z 393.438,A -85,B 0,C 180,E1 20551.293,E2 20551.293} C_VEL
LIN {X 0,Y 426.976,Z 391.43,A -85,B 0,C 180,E1 20550.931,E2 20550.931} C_VEL
LIN {X 0,Y 423.886,Z 388.457,A -85,B 0,C 180,E1 20550.122,E2 20550.122} C_VEL
LIN {X 0,Y 422.117,Z 385.352,A -85,B 0,C 180,E1 20549.595,E2 20549.595} C_VEL
LIN {X 0,Y 419.092,Z 383.1,A -85,B 0,C 180,E1 20548.773,E2 20548.773} C_VEL
LIN {X 0,Y 417.617,Z 380.298,A -85,B 0,C 180,E1 20548.298,E2 20548.298} C_VEL
LIN {X 0,Y 417.358,Z 379.021,A -85,B 0,C 180,E1 20548.161,E2 20548.161} C_VEL
LIN {X 0,Y 417.334,Z 379.016,A -85,B 0,C 180,E1 20544.451,E2 20544.451} C_VEL
LIN {X 0,Y 417.337,Z 379.063,A -85,B 0,C 180,E1 20540.621,E2 20540.621} C_VEL
LIN {X 0,Y 417.338,Z 379.005,A -85,B 0,C 180,E1 20536.852,E2 20536.852} C_VEL
LIN {X 0,Y 417.371,Z 379.055,A -85,B 0,C 180,E1 20533.155,E2 20533.155} C_VEL
LIN {X 0,Y 417.369,Z 379.051,A -85,B 0,C 180,E1 20529.237,E2 20529.237} C_VEL
LIN {X 0,Y 417.34,Z 379.054,A -85,B 0,C 180,E1 20525.499,E2 20525.499} C_VEL
LIN {X 0,Y 417.315,Z 379.056,A -85,B 0,C 180,E1 20521.785,E2 20521.785} C_VEL
LIN {X 0,Y 417.306,Z 379.054,A -85,B 0,C 180,E1 20517.941,E2 20517.941} C_VEL
LIN {X 0,Y 417.307,Z 379.051,A -85,B 0,C 180,E1 20514.087,E2 20514.087} C_VEL
LIN {X 0,Y 417.338,Z 379.049,A -85,B 0,C 180,E1 20510.485,E2 20510.485} C_VEL
LIN {X 0,Y 417.359,Z 379.05,A -85,B 0,C 180,E1 20506.542,E2 20506.542} C_VEL
LIN {X 0,Y 417.341,Z 379.012,A -85,B 0,C 180,E1 20502.718,E2 20502.718} C_VEL
LIN {X 0,Y 417.327,Z 379.066,A -85,B 0,C 180,E1 20498.938,E2 20498.938} C_VEL
LIN {X 0,Y 417.316,Z 379.026,A -85,B 0,C 180,E1 20495.211,E2 20495.211} C_VEL
LIN {X 0,Y 417.344,Z 379.144,A -85,B 0,C 180,E1 20492.823,E2 20492.823} C_VEL
LIN {X 0,Y 418.692,Z 382.555,A -85,B 0,C 180,E1 20491.937,E2 20491.937} C_VEL
LIN {X 0,Y 420.847,Z 385.122,A -85,B 0,C 180,E1 20491.204,E2 20491.204} C_VEL
LIN {X 0,Y 423.861,Z 389.122,A -85,B 0,C 180,E1 20490.345,E2 20490.345} C_VEL
LIN {X 0,Y 425.536,Z 391.073,A -85,B 0,C 180,E1 20489.891,E2 20489.891} C_VEL
LIN {X 0,Y 429.034,Z 395.537,A -85,B 0,C 180,E1 20488.962,E2 20488.962} C_VEL
LIN {X 0,Y 437.847,Z 407.351,A -85,B 0,C 180,E1 20486.766,E2 20486.766} C_VEL
LIN {X 0,Y 447.362,Z 420.486,A -85,B 0,C 180,E1 20484.61,E2 20484.61} C_VEL
LIN {X 0,Y 458.989,Z 437.881,A -85,B 0,C 180,E1 20482.198,E2 20482.198} C_VEL
LIN {X 0,Y 466.874,Z 450.748,A -85,B 0,C 180,E1 20480.673,E2 20480.673} C_VEL
LIN {X 0,Y 459.663,Z 657.326,A -85,B 0,C 180,E1 20476.942,E2 20476.942} C_VEL
LIN {X 0,Y 456.8,Z 738.47,A -85,B 0,C 180,E1 20475.466,E2 20475.466} C_VEL
LIN {X 0,Y 454.92,Z 761.917,A -85,B 0,C 180,E1 20474.854,E2 20474.854} C_VEL
LIN {X 0,Y 452.624,Z 784.585,A -85,B 0,C 180,E1 20474.044,E2 20474.044} C_VEL
LIN {X 0,Y 450.008,Z 805.085,A -85,B 0,C 180,E1 20473.09,E2 20473.09} C_VEL
LIN {X 0,Y 446.978,Z 826.333,A -85,B 0,C 180,E1 20471.886,E2 20471.886} C_VEL
LIN {X 0,Y 443.604,Z 846.742,A -85,B 0,C 180,E1 20470.471,E2 20470.471} C_VEL
LIN {X 0,Y 439.977,Z 867.277,A -85,B 0,C 180,E1 20468.788,E2 20468.788} C_VEL
LIN {X 0,Y 436.484,Z 885.784,A -85,B 0,C 180,E1 20466.991,E2 20466.991} C_VEL
LIN {X 0,Y 432.631,Z 905.593,A -85,B 0,C 180,E1 20464.741,E2 20464.741} C_VEL
LIN {X 0,Y 429.376,Z 922.264,A -85,B 0,C 180,E1 20462.538,E2 20462.538} C_VEL
LIN {X 0,Y 426.236,Z 938.425,A -85,B 0,C 180,E1 20460.05,E2 20460.05} C_VEL
LIN {X 0,Y 423.513,Z 953.364,A -85,B 0,C 180,E1 20457.408,E2 20457.408} C_VEL
LIN {X 0,Y 421.155,Z 966.88,A -85,B 0,C 180,E1 20454.596,E2 20454.596} C_VEL
LIN {X 0,Y 419.229,Z 979.456,A -85,B 0,C 180,E1 20451.543,E2 20451.543} C_VEL
LIN {X 0,Y 417.932,Z 989.382,A -85,B 0,C 180,E1 20448.696,E2 20448.696} C_VEL
LIN {X 0,Y 417,Z 997.994,A -85,B 0,C 180,E1 20445.719,E2 20445.719} C_VEL
LIN {X 0,Y 416.426,Z 1004.595,A -85,B 0,C 180,E1 20442.886,E2 20442.886} C_VEL
LIN {X 0,Y 416.069,Z 1010.43,A -85,B 0,C 180,E1 20439.683,E2 20439.683} C_VEL
LIN {X 0,Y 415.937,Z 1013.959,A -85,B 0,C 180,E1 20437.042,E2 20437.042} C_VEL
LIN {X 0,Y 415.91,Z 1016.712,A -85,B 0,C 180,E1 20433.998,E2 20433.998} C_VEL
LIN {X 0,Y 415.897,Z 1017.825,A -85,B 0,C 180,E1 20431.102,E2 20431.102} C_VEL
LIN {X 0,Y 415.906,Z 1017.735,A -85,B 0,C 180,E1 20428.347,E2 20428.347} C_VEL
LIN {X 0,Y 415.911,Z 1016.068,A -85,B 0,C 180,E1 20425.174,E2 20425.174} C_VEL
LIN {X 0,Y 415.952,Z 1013.48,A -85,B 0,C 180,E1 20422.543,E2 20422.543} C_VEL
LIN {X 0,Y 416.138,Z 1009.101,A -85,B 0,C 180,E1 20419.48,E2 20419.48} C_VEL
LIN {X 0,Y 416.52,Z 1003.35,A -85,B 0,C 180,E1 20416.537,E2 20416.537} C_VEL
LIN {X 0,Y 417.258,Z 995.362,A -85,B 0,C 180,E1 20413.291,E2 20413.291} C_VEL
LIN {X 0,Y 418.214,Z 987.041,A -85,B 0,C 180,E1 20410.593,E2 20410.593} C_VEL
LIN {X 0,Y 419.798,Z 975.573,A -85,B 0,C 180,E1 20407.455,E2 20407.455} C_VEL
LIN {X 0,Y 421.663,Z 963.864,A -85,B 0,C 180,E1 20404.738,E2 20404.738} C_VEL
LIN {X 0,Y 424.171,Z 949.479,A -85,B 0,C 180,E1 20401.876,E2 20401.876} C_VEL
LIN {X 0,Y 427.119,Z 933.991,A -85,B 0,C 180,E1 20399.217,E2 20399.217} C_VEL
LIN {X 0,Y 430.264,Z 917.642,A -85,B 0,C 180,E1 20396.825,E2 20396.825} C_VEL
LIN {X 0,Y 433.872,Z 899.328,A -85,B 0,C 180,E1 20394.503,E2 20394.503} C_VEL
LIN {X 0,Y 437.329,Z 881.317,A -85,B 0,C 180,E1 20392.55,E2 20392.55} C_VEL
LIN {X 0,Y 441.216,Z 860.416,A -85,B 0,C 180,E1 20390.622,E2 20390.622} C_VEL
LIN {X 0,Y 444.541,Z 841.299,A -85,B 0,C 180,E1 20389.123,E2 20389.123} C_VEL
LIN {X 0,Y 447.931,Z 819.571,A -85,B 0,C 180,E1 20387.707,E2 20387.707} C_VEL
LIN {X 0,Y 450.994,Z 797.949,A -85,B 0,C 180,E1 20386.548,E2 20386.548} C_VEL
LIN {X 0,Y 453.523,Z 776.216,A -85,B 0,C 180,E1 20385.637,E2 20385.637} C_VEL
LIN {X 0,Y 455.718,Z 753.554,A -85,B 0,C 180,E1 20384.902,E2 20384.902} C_VEL
LIN {X 0,Y 457.159,Z 730.786,A -85,B 0,C 180,E1 20384.382,E2 20384.382} C_VEL
LIN {X 0,Y 464.143,Z 526.022,A -85,B 0,C 180,E1 20380.695,E2 20380.695} C_VEL
LIN {X 0,Y 466.768,Z 450.446,A -85,B 0,C 180,E1 20379.31,E2 20379.31} C_VEL
LIN {X 0,Y 455.694,Z 432.9,A -85,B 0,C 180,E1 20377.152,E2 20377.152} C_VEL
LIN {X 0,Y 444.223,Z 416.056,A -85,B 0,C 180,E1 20374.712,E2 20374.712} C_VEL
LIN {X 0,Y 435.27,Z 403.907,A -85,B 0,C 180,E1 20372.632,E2 20372.632} C_VEL
LIN {X 0,Y 428.501,Z 395.016,A -85,B 0,C 180,E1 20370.925,E2 20370.925} C_VEL
LIN {X 0,Y 425.154,Z 390.401,A -85,B 0,C 180,E1 20370.022,E2 20370.022} C_VEL
LIN {X 0,Y 421.291,Z 385.904,A -85,B 0,C 180,E1 20368.957,E2 20368.957} C_VEL
LIN {X 0,Y 420.03,Z 384.08,A -85,B 0,C 180,E1 20368.585,E2 20368.585} C_VEL
LIN {X 0,Y 417.899,Z 381.062,A -85,B 0,C 180,E1 20367.655,E2 20367.655} C_VEL
LIN {X 0,Y 417.333,Z 379.044,A -85,B 0,C 180,E1 20367.18,E2 20367.18} C_VEL
LIN {X 0,Y 417.352,Z 379.005,A -85,B 0,C 180,E1 20363.433,E2 20363.433} C_VEL
LIN {X 0,Y 417.358,Z 379.039,A -85,B 0,C 180,E1 20359.714,E2 20359.714} C_VEL
LIN {X 0,Y 417.332,Z 379.028,A -85,B 0,C 180,E1 20355.85,E2 20355.85} C_VEL
LIN {X 0,Y 417.307,Z 379.053,A -85,B 0,C 180,E1 20352.172,E2 20352.172} C_VEL
LIN {X 0,Y 417.3,Z 379.059,A -85,B 0,C 180,E1 20348.336,E2 20348.336} C_VEL
LIN {X 0,Y 417.309,Z 379.061,A -85,B 0,C 180,E1 20344.535,E2 20344.535} C_VEL
LIN {X 0,Y 417.342,Z 379.057,A -85,B 0,C 180,E1 20340.823,E2 20340.823} C_VEL
LIN {X 0,Y 417.356,Z 379.058,A -85,B 0,C 180,E1 20336.979,E2 20336.979} C_VEL
LIN {X 0,Y 417.351,Z 379.061,A -85,B 0,C 180,E1 20333.12,E2 20333.12} C_VEL
LIN {X 0,Y 417.329,Z 379.064,A -85,B 0,C 180,E1 20329.369,E2 20329.369} C_VEL
LIN {X 0,Y 417.324,Z 379.065,A -85,B 0,C 180,E1 20325.571,E2 20325.571} C_VEL
LIN {X 0,Y 417.324,Z 379.012,A -85,B 0,C 180,E1 20321.708,E2 20321.708} C_VEL
LIN {X 0,Y 417.343,Z 379.033,A -85,B 0,C 180,E1 20317.905,E2 20317.905} C_VEL
LIN {X 0,Y 417.37,Z 379.037,A -85,B 0,C 180,E1 20314.151,E2 20314.151} C_VEL
LIN {X 0,Y 417.375,Z 379.226,A -85,B 0,C 180,E1 20311.684,E2 20311.684} C_VEL
LIN {X 0,Y 418.367,Z 382.072,A -85,B 0,C 180,E1 20311.329,E2 20311.329} C_VEL
LIN {X 0,Y 420.852,Z 384.676,A -85,B 0,C 180,E1 20310.62,E2 20310.62} C_VEL
LIN {X 0,Y 422.447,Z 385.785,A -85,B 0,C 180,E1 20310.196,E2 20310.196} C_VEL
LIN {X 0,Y 424.668,Z 389.459,A -85,B 0,C 180,E1 20309.549,E2 20309.549} C_VEL
LIN {X 0,Y 427.558,Z 392.163,A -85,B 0,C 180,E1 20308.803,E2 20308.803} C_VEL
LIN {X 0,Y 430.51,Z 396.226,A -85,B 0,C 180,E1 20308.026,E2 20308.026} C_VEL
LIN {X 0,Y 432.489,Z 398.237,A -85,B 0,C 180,E1 20307.542,E2 20307.542} C_VEL
LIN {X 0,Y 436.125,Z 402.753,A -85,B 0,C 180,E1 20306.657,E2 20306.657} C_VEL
LIN {X 0,Y 442.505,Z 411.124,A -85,B 0,C 180,E1 20305.173,E2 20305.173} C_VEL
LIN {X 0,Y 449.029,Z 419.461,A -85,B 0,C 180,E1 20303.758,E2 20303.758} C_VEL
LIN {X 0,Y 460.316,Z 435.14,A -85,B 0,C 180,E1 20301.475,E2 20301.475} C_VEL
LIN {X 0,Y 466.685,Z 444.69,A -85,B 0,C 180,E1 20300.266,E2 20300.266} C_VEL
LIN {X 0,Y 459.543,Z 647.414,A -85,B 0,C 180,E1 20296.603,E2 20296.603} C_VEL
LIN {X 0,Y 457.084,Z 715.107,A -85,B 0,C 180,E1 20295.365,E2 20295.365} C_VEL
LIN {X 0,Y 455.379,Z 737.538,A -85,B 0,C 180,E1 20294.757,E2 20294.757} C_VEL
LIN {X 0,Y 453.269,Z 759.372,A -85,B 0,C 180,E1 20293.965,E2 20293.965} C_VEL
LIN {X 0,Y 452.005,Z 769.58,A -85,B 0,C 180,E1 20293.511,E2 20293.511} C_VEL
LIN {X 0,Y 450.396,Z 776.917,A -85,B 0,C 180,E1 20293.253,E2 20293.253} C_VEL
LIN {X 0,Y 443.421,Z 795.388,A -85,B 0,C 180,E1 20292.773,E2 20292.773} C_VEL
LIN {X 0,Y 441.503,Z 802.364,A -85,B 0,C 180,E1 20292.417,E2 20292.417} C_VEL
LIN {X 0,Y 438.038,Z 822.132,A -85,B 0,C 180,E1 20291.008,E2 20291.008} C_VEL
LIN {X 0,Y 434.179,Z 842.44,A -85,B 0,C 180,E1 20289.287,E2 20289.287} C_VEL
LIN {X 0,Y 430.621,Z 859.814,A -85,B 0,C 180,E1 20287.548,E2 20287.548} C_VEL
LIN {X 0,Y 426.594,Z 878.623,A -85,B 0,C 180,E1 20285.348,E2 20285.348} C_VEL
LIN {X 0,Y 423.08,Z 894.633,A -85,B 0,C 180,E1 20283.163,E2 20283.163} C_VEL
LIN {X 0,Y 419.626,Z 910.396,A -85,B 0,C 180,E1 20280.653,E2 20280.653} C_VEL
LIN {X 0,Y 416.644,Z 924.526,A -85,B 0,C 180,E1 20278.054,E2 20278.054} C_VEL
LIN {X 0,Y 414.057,Z 937.249,A -85,B 0,C 180,E1 20275.3,E2 20275.3} C_VEL
LIN {X 0,Y 411.952,Z 948.938,A -85,B 0,C 180,E1 20272.371,E2 20272.371} C_VEL
LIN {X 0,Y 410.328,Z 958.971,A -85,B 0,C 180,E1 20269.351,E2 20269.351} C_VEL
LIN {X 0,Y 409.179,Z 967.814,A -85,B 0,C 180,E1 20266.172,E2 20266.172} C_VEL
LIN {X 0,Y 408.494,Z 974.57,A -85,B 0,C 180,E1 20263.156,E2 20263.156} C_VEL
LIN {X 0,Y 408.076,Z 980.573,A -85,B 0,C 180,E1 20259.732,E2 20259.732} C_VEL
LIN {X 0,Y 407.939,Z 984.068,A -85,B 0,C 180,E1 20257.038,E2 20257.038} C_VEL
LIN {X 0,Y 407.913,Z 986.757,A -85,B 0,C 180,E1 20253.935,E2 20253.935} C_VEL
LIN {X 0,Y 407.901,Z 987.818,A -85,B 0,C 180,E1 20251.123,E2 20251.123} C_VEL
LIN {X 0,Y 407.907,Z 987.742,A -85,B 0,C 180,E1 20248.314,E2 20248.314} C_VEL
LIN {X 0,Y 407.912,Z 986.104,A -85,B 0,C 180,E1 20245.079,E2 20245.079} C_VEL
LIN {X 0,Y 407.958,Z 983.531,A -85,B 0,C 180,E1 20242.395,E2 20242.395} C_VEL
LIN {X 0,Y 408.163,Z 979.18,A -85,B 0,C 180,E1 20239.271,E2 20239.271} C_VEL
LIN {X 0,Y 408.577,Z 973.574,A -85,B 0,C 180,E1 20236.27,E2 20236.27} C_VEL
LIN {X 0,Y 409.359,Z 966.218,A -85,B 0,C 180,E1 20233.104,E2 20233.104} C_VEL
LIN {X 0,Y 410.477,Z 957.894,A -85,B 0,C 180,E1 20230.211,E2 20230.211} C_VEL
LIN {X 0,Y 412.178,Z 947.52,A -85,B 0,C 180,E1 20227.164,E2 20227.164} C_VEL
LIN {X 0,Y 414.23,Z 936.365,A -85,B 0,C 180,E1 20224.404,E2 20224.404} C_VEL
LIN {X 0,Y 417.15,Z 921.934,A -85,B 0,C 180,E1 20221.359,E2 20221.359} C_VEL
LIN {X 0,Y 420.275,Z 907.539,A -85,B 0,C 180,E1 20218.763,E2 20218.763} C_VEL
LIN {X 0,Y 423.718,Z 891.689,A -85,B 0,C 180,E1 20216.325,E2 20216.325} C_VEL
LIN {X 0,Y 427.5,Z 874.639,A -85,B 0,C 180,E1 20214.056,E2 20214.056} C_VEL
LIN {X 0,Y 431.275,Z 856.633,A -85,B 0,C 180,E1 20212.022,E2 20212.022} C_VEL
LIN {X 0,Y 435.341,Z 836.581,A -85,B 0,C 180,E1 20210.095,E2 20210.095} C_VEL
LIN {X 0,Y 438.698,Z 818.604,A -85,B 0,C 180,E1 20208.633,E2 20208.633} C_VEL
LIN {X 0,Y 442.386,Z 796.688,A -85,B 0,C 180,E1 20207.138,E2 20207.138} C_VEL
LIN {X 0,Y 445.213,Z 777.533,A -85,B 0,C 180,E1 20206.062,E2 20206.062} C_VEL
LIN {X 0,Y 448.089,Z 754.051,A -85,B 0,C 180,E1 20205.005,E2 20205.005} C_VEL
LIN {X 0,Y 450.34,Z 731.39,A -85,B 0,C 180,E1 20204.228,E2 20204.228} C_VEL
LIN {X 0,Y 451.866,Z 708.414,A -85,B 0,C 180,E1 20203.68,E2 20203.68} C_VEL
LIN {X 0,Y 459.38,Z 503.886,A -85,B 0,C 180,E1 20199.956,E2 20199.956} C_VEL
LIN {X 0,Y 461.454,Z 448.31,A -85,B 0,C 180,E1 20198.929,E2 20198.929} C_VEL
LIN {X 0,Y 448.922,Z 430.278,A -85,B 0,C 180,E1 20196.41,E2 20196.41} C_VEL
LIN {X 0,Y 440.006,Z 418.578,A -85,B 0,C 180,E1 20194.46,E2 20194.46} C_VEL
LIN {X 0,Y 435.956,Z 413.339,A -85,B 0,C 180,E1 20193.515,E2 20193.515} C_VEL
LIN {X 0,Y 432.483,Z 408.874,A -85,B 0,C 180,E1 20192.672,E2 20192.672} C_VEL
LIN {X 0,Y 428.505,Z 403.894,A -85,B 0,C 180,E1 20191.669,E2 20191.669} C_VEL
LIN {X 0,Y 425.09,Z 399.653,A -85,B 0,C 180,E1 20190.77,E2 20190.77} C_VEL
LIN {X 0,Y 423.737,Z 398.119,A -85,B 0,C 180,E1 20190.407,E2 20190.407} C_VEL
LIN {X 0,Y 420.571,Z 394.417,A -85,B 0,C 180,E1 20189.53,E2 20189.53} C_VEL
LIN {X 0,Y 419.396,Z 392.573,A -85,B 0,C 180,E1 20189.179,E2 20189.179} C_VEL
LIN {X 0,Y 416.246,Z 389.713,A -85,B 0,C 180,E1 20188.282,E2 20188.282} C_VEL
LIN {X 0,Y 414.39,Z 386.447,A -85,B 0,C 180,E1 20187.676,E2 20187.676} C_VEL
LIN {X 0,Y 411.331,Z 384.336,A -85,B 0,C 180,E1 20186.763,E2 20186.763} C_VEL
LIN {X 0,Y 409.756,Z 381.569,A -85,B 0,C 180,E1 20186.21,E2 20186.21} C_VEL
LIN {X 0,Y 409.424,Z 380.042,A -85,B 0,C 180,E1 20186.025,E2 20186.025} C_VEL
LIN {X 0,Y 409.398,Z 380.007,A -85,B 0,C 180,E1 20182.244,E2 20182.244} C_VEL
LIN {X 0,Y 409.39,Z 380.008,A -85,B 0,C 180,E1 20178.512,E2 20178.512} C_VEL
LIN {X 0,Y 409.397,Z 380.033,A -85,B 0,C 180,E1 20174.714,E2 20174.714} C_VEL
LIN {X 0,Y 409.418,Z 380.04,A -85,B 0,C 180,E1 20170.982,E2 20170.982} C_VEL
LIN {X 0,Y 409.44,Z 380.041,A -85,B 0,C 180,E1 20167.155,E2 20167.155} C_VEL
LIN {X 0,Y 409.414,Z 380.048,A -85,B 0,C 180,E1 20163.22,E2 20163.22} C_VEL
LIN {X 0,Y 409.386,Z 380.052,A -85,B 0,C 180,E1 20159.441,E2 20159.441} C_VEL
LIN {X 0,Y 409.367,Z 380.054,A -85,B 0,C 180,E1 20155.658,E2 20155.658} C_VEL
LIN {X 0,Y 409.362,Z 380.054,A -85,B 0,C 180,E1 20151.715,E2 20151.715} C_VEL
LIN {X 0,Y 409.365,Z 380.046,A -85,B 0,C 180,E1 20147.732,E2 20147.732} C_VEL
LIN {X 0,Y 409.381,Z 380.023,A -85,B 0,C 180,E1 20143.98,E2 20143.98} C_VEL
LIN {X 0,Y 409.408,Z 380.03,A -85,B 0,C 180,E1 20140.156,E2 20140.156} C_VEL
LIN {X 0,Y 409.424,Z 379.999,A -85,B 0,C 180,E1 20136.304,E2 20136.304} C_VEL
LIN {X 0,Y 409.396,Z 380.047,A -85,B 0,C 180,E1 20134.796,E2 20134.796} C_VEL
LIN {X 0,Y 410.713,Z 383.521,A -85,B 0,C 180,E1 20133.924,E2 20133.924} C_VEL
LIN {X 0,Y 413.336,Z 385.996,A -85,B 0,C 180,E1 20133.106,E2 20133.106} C_VEL
LIN {X 0,Y 416.579,Z 390.294,A -85,B 0,C 180,E1 20132.094,E2 20132.094} C_VEL
LIN {X 0,Y 418.362,Z 392.392,A -85,B 0,C 180,E1 20131.567,E2 20131.567} C_VEL
LIN {X 0,Y 422.035,Z 396.918,A -85,B 0,C 180,E1 20130.516,E2 20130.516} C_VEL
LIN {X 0,Y 426.24,Z 402.452,A -85,B 0,C 180,E1 20129.362,E2 20129.362} C_VEL
LIN {X 0,Y 434.938,Z 414.281,A -85,B 0,C 180,E1 20127.145,E2 20127.145} C_VEL
LIN {X 0,Y 444.091,Z 427.095,A -85,B 0,C 180,E1 20125.021,E2 20125.021} C_VEL
LIN {X 0,Y 455.24,Z 443.96,A -85,B 0,C 180,E1 20122.651,E2 20122.651} C_VEL
LIN {X 0,Y 461.653,Z 454.487,A -85,B 0,C 180,E1 20121.372,E2 20121.372} C_VEL
LIN {X 0,Y 454.093,Z 660.23,A -85,B 0,C 180,E1 20117.626,E2 20117.626} C_VEL
LIN {X 0,Y 451.187,Z 738.292,A -85,B 0,C 180,E1 20116.192,E2 20116.192} C_VEL
LIN {X 0,Y 449.237,Z 761.625,A -85,B 0,C 180,E1 20115.58,E2 20115.58} C_VEL
LIN {X 0,Y 446.825,Z 784.287,A -85,B 0,C 180,E1 20114.768,E2 20114.768} C_VEL
LIN {X 0,Y 444.083,Z 804.784,A -85,B 0,C 180,E1 20113.81,E2 20113.81} C_VEL
LIN {X 0,Y 440.906,Z 826.028,A -85,B 0,C 180,E1 20112.598,E2 20112.598} C_VEL
LIN {X 0,Y 437.369,Z 846.437,A -85,B 0,C 180,E1 20111.172,E2 20111.172} C_VEL
LIN {X 0,Y 433.649,Z 866.505,A -85,B 0,C 180,E1 20109.517,E2 20109.517} C_VEL
LIN {X 0,Y 429.804,Z 885.734,A -85,B 0,C 180,E1 20107.632,E2 20107.632} C_VEL
LIN {X 0,Y 425.769,Z 905.393,A -85,B 0,C 180,E1 20105.367,E2 20105.367} C_VEL
LIN {X 0,Y 422.328,Z 921.949,A -85,B 0,C 180,E1 20103.15,E2 20103.15} C_VEL
LIN {X 0,Y 419.088,Z 937.675,A -85,B 0,C 180,E1 20100.698,E2 20100.698} C_VEL
LIN {X 0,Y 416.211,Z 952.297,A -85,B 0,C 180,E1 20098.086,E2 20098.086} C_VEL
LIN {X 0,Y 413.748,Z 965.487,A -85,B 0,C 180,E1 20095.321,E2 20095.321} C_VEL
LIN {X 0,Y 411.756,Z 977.554,A -85,B 0,C 180,E1 20092.408,E2 20092.408} C_VEL
LIN {X 0,Y 410.209,Z 988.132,A -85,B 0,C 180,E1 20089.357,E2 20089.357} C_VEL
LIN {X 0,Y 409.123,Z 997.408,A -85,B 0,C 180,E1 20086.169,E2 20086.169} C_VEL
LIN {X 0,Y 408.502,Z 1004.183,A -85,B 0,C 180,E1 20083.3,E2 20083.3} C_VEL
LIN {X 0,Y 408.118,Z 1009.811,A -85,B 0,C 180,E1 20080.302,E2 20080.302} C_VEL
LIN {X 0,Y 407.952,Z 1013.64,A -85,B 0,C 180,E1 20077.463,E2 20077.463} C_VEL
LIN {X 0,Y 407.909,Z 1016.295,A -85,B 0,C 180,E1 20074.64,E2 20074.64} C_VEL
LIN {X 0,Y 407.907,Z 1017.78,A -85,B 0,C 180,E1 20071.405,E2 20071.405} C_VEL
LIN {X 0,Y 407.904,Z 1017.802,A -85,B 0,C 180,E1 20068.736,E2 20068.736} C_VEL
LIN {X 0,Y 407.91,Z 1016.522,A -85,B 0,C 180,E1 20065.643,E2 20065.643} C_VEL
LIN {X 0,Y 407.947,Z 1013.799,A -85,B 0,C 180,E1 20062.679,E2 20062.679} C_VEL
LIN {X 0,Y 408.103,Z 1010.019,A -85,B 0,C 180,E1 20059.841,E2 20059.841} C_VEL
LIN {X 0,Y 408.478,Z 1004.495,A -85,B 0,C 180,E1 20056.844,E2 20056.844} C_VEL
LIN {X 0,Y 409.087,Z 997.755,A -85,B 0,C 180,E1 20053.97,E2 20053.97} C_VEL
LIN {X 0,Y 410.151,Z 988.607,A -85,B 0,C 180,E1 20050.789,E2 20050.789} C_VEL
LIN {X 0,Y 411.581,Z 978.616,A -85,B 0,C 180,E1 20047.883,E2 20047.883} C_VEL
LIN {X 0,Y 413.634,Z 966.142,A -85,B 0,C 180,E1 20044.825,E2 20044.825} C_VEL
LIN {X 0,Y 416.071,Z 953.053,A -85,B 0,C 180,E1 20042.06,E2 20042.06} C_VEL
LIN {X 0,Y 418.909,Z 938.54,A -85,B 0,C 180,E1 20039.448,E2 20039.448} C_VEL
LIN {X 0,Y 422.157,Z 922.836,A -85,B 0,C 180,E1 20036.974,E2 20036.974} C_VEL
LIN {X 0,Y 425.647,Z 905.963,A -85,B 0,C 180,E1 20034.705,E2 20034.705} C_VEL
LIN {X 0,Y 429.472,Z 887.462,A -85,B 0,C 180,E1 20032.549,E2 20032.549} C_VEL
LIN {X 0,Y 433.183,Z 868.727,A -85,B 0,C 180,E1 20030.69,E2 20030.69} C_VEL
LIN {X 0,Y 437.206,Z 847.344,A -85,B 0,C 180,E1 20028.897,E2 20028.897} C_VEL
LIN {X 0,Y 440.485,Z 828.438,A -85,B 0,C 180,E1 20027.563,E2 20027.563} C_VEL
LIN {X 0,Y 443.902,Z 806.061,A -85,B 0,C 180,E1 20026.258,E2 20026.258} C_VEL
LIN {X 0,Y 446.72,Z 785.007,A -85,B 0,C 180,E1 20025.265,E2 20025.265} C_VEL
LIN {X 0,Y 449.179,Z 762.108,A -85,B 0,C 180,E1 20024.436,E2 20024.436} C_VEL
LIN {X 0,Y 451.152,Z 738.747,A -85,B 0,C 180,E1 20023.818,E2 20023.818} C_VEL
LIN {X 0,Y 453.811,Z 667.782,A -85,B 0,C 180,E1 20022.512,E2 20022.512} C_VEL
LIN {X 0,Y 461.277,Z 463.601,A -85,B 0,C 180,E1 20018.797,E2 20018.797} C_VEL
LIN {X 0,Y 461.518,Z 454.089,A -85,B 0,C 180,E1 20018.604,E2 20018.604} C_VEL
LIN {X 0,Y 449.724,Z 435.521,A -85,B 0,C 180,E1 20016.216,E2 20016.216} C_VEL
LIN {X 0,Y 439.867,Z 421.162,A -85,B 0,C 180,E1 20014.038,E2 20014.038} C_VEL
LIN {X 0,Y 430.069,Z 407.522,A -85,B 0,C 180,E1 20011.657,E2 20011.657} C_VEL
LIN {X 0,Y 424.803,Z 400.872,A -85,B 0,C 180,E1 20010.283,E2 20010.283} C_VEL
LIN {X 0,Y 421.626,Z 396.533,A -85,B 0,C 180,E1 20009.398,E2 20009.398} C_VEL
LIN {X 0,Y 418.199,Z 392.126,A -85,B 0,C 180,E1 20008.41,E2 20008.41} C_VEL
LIN {X 0,Y 413.744,Z 386.658,A -85,B 0,C 180,E1 20007.06,E2 20007.06} C_VEL
LIN {X 0,Y 412.403,Z 385.367,A -85,B 0,C 180,E1 20006.649,E2 20006.649} C_VEL
LIN {X 0,Y 410.14,Z 382.48,A -85,B 0,C 180,E1 20005.872,E2 20005.872} C_VEL
LIN {X 0,Y 409.394,Z 380.011,A -85,B 0,C 180,E1 20005.205,E2 20005.205} C_VEL
LIN {X 0,Y 409.424,Z 380.027,A -85,B 0,C 180,E1 20001.488,E2 20001.488} C_VEL
LIN {X 0,Y 409.412,Z 379.99,A -85,B 0,C 180,E1 19997.627,E2 19997.627} C_VEL
LIN {X 0,Y 409.39,Z 380.052,A -85,B 0,C 180,E1 19993.848,E2 19993.848} C_VEL
LIN {X 0,Y 409.367,Z 380.051,A -85,B 0,C 180,E1 19990.128,E2 19990.128} C_VEL
LIN {X 0,Y 409.36,Z 380.047,A -85,B 0,C 180,E1 19986.294,E2 19986.294} C_VEL
LIN {X 0,Y 409.368,Z 380.041,A -85,B 0,C 180,E1 19982.379,E2 19982.379} C_VEL
LIN {X 0,Y 409.391,Z 380.038,A -85,B 0,C 180,E1 19978.6,E2 19978.6} C_VEL
LIN {X 0,Y 409.419,Z 380.035,A -85,B 0,C 180,E1 19974.815,E2 19974.815} C_VEL
LIN {X 0,Y 409.416,Z 380.036,A -85,B 0,C 180,E1 19971.008,E2 19971.008} C_VEL
LIN {X 0,Y 409.399,Z 380.038,A -85,B 0,C 180,E1 19967.159,E2 19967.159} C_VEL
LIN {X 0,Y 409.384,Z 380,A -85,B 0,C 180,E1 19963.396,E2 19963.396} C_VEL
LIN {X 0,Y 409.393,Z 380.052,A -85,B 0,C 180,E1 19959.558,E2 19959.558} C_VEL
LIN {X 0,Y 409.398,Z 379.997,A -85,B 0,C 180,E1 19955.776,E2 19955.776} C_VEL
LIN {X 0,Y 409.441,Z 380.248,A -85,B 0,C 180,E1 19953.807,E2 19953.807} C_VEL
LIN {X 0,Y 410.444,Z 383.123,A -85,B 0,C 180,E1 19953.409,E2 19953.409} C_VEL
LIN {X 0,Y 412.755,Z 385.592,A -85,B 0,C 180,E1 19952.674,E2 19952.674} C_VEL
LIN {X 0,Y 414.683,Z 386.853,A -85,B 0,C 180,E1 19952.111,E2 19952.111} C_VEL
LIN {X 0,Y 416.761,Z 390.375,A -85,B 0,C 180,E1 19951.443,E2 19951.443} C_VEL
LIN {X 0,Y 419.83,Z 393.095,A -85,B 0,C 180,E1 19950.58,E2 19950.58} C_VEL
LIN {X 0,Y 422.609,Z 397.085,A -85,B 0,C 180,E1 19949.778,E2 19949.778} C_VEL
LIN {X 0,Y 424.927,Z 399.409,A -85,B 0,C 180,E1 19949.164,E2 19949.164} C_VEL
LIN {X 0,Y 428.408,Z 403.824,A -85,B 0,C 180,E1 19948.244,E2 19948.244} C_VEL
LIN {X 0,Y 430.27,Z 406.134,A -85,B 0,C 180,E1 19947.77,E2 19947.77} C_VEL
LIN {X 0,Y 434.786,Z 411.827,A -85,B 0,C 180,E1 19946.659,E2 19946.659} C_VEL
LIN {X 0,Y 439.427,Z 417.857,A -85,B 0,C 180,E1 19945.568,E2 19945.568} C_VEL
LIN {X 0,Y 446.381,Z 426.99,A -85,B 0,C 180,E1 19944.026,E2 19944.026} C_VEL
LIN {X 0,Y 456.774,Z 441.539,A -85,B 0,C 180,E1 19941.882,E2 19941.882} C_VEL
LIN {X 0,Y 461.469,Z 448.702,A -85,B 0,C 180,E1 19940.962,E2 19940.962} C_VEL
LIN {X 0,Y 453.873,Z 653.716,A -85,B 0,C 180,E1 19937.229,E2 19937.229} C_VEL
LIN {X 0,Y 451.479,Z 715.857,A -85,B 0,C 180,E1 19936.078,E2 19936.078} C_VEL
LIN {X 0,Y 449.676,Z 738.373,A -85,B 0,C 180,E1 19935.459,E2 19935.459} C_VEL
LIN {X 0,Y 447.423,Z 760.437,A -85,B 0,C 180,E1 19934.646,E2 19934.646} C_VEL
LIN {X 0,Y 444.854,Z 780.05,A -85,B 0,C 180,E1 19933.714,E2 19933.714} C_VEL
LIN {X 0,Y 441.892,Z 800.017,A -85,B 0,C 180,E1 19932.567,E2 19932.567} C_VEL
LIN {X 0,Y 441.503,Z 802.364,A -85,B 0,C 180,E1 19932.417,E2 19932.417} C_VEL
LIN {X 0,Y 439.526,Z 809.4,A -85,B 0,C 180,E1 19932.035,E2 19932.035} C_VEL
LIN {X 0,Y 431.831,Z 827.037,A -85,B 0,C 180,E1 19931.268,E2 19931.268} C_VEL
LIN {X 0,Y 429.779,Z 833.515,A -85,B 0,C 180,E1 19930.804,E2 19930.804} C_VEL
LIN {X 0,Y 425.781,Z 852.872,A -85,B 0,C 180,E1 19928.996,E2 19928.996} C_VEL
LIN {X 0,Y 421.771,Z 870.701,A -85,B 0,C 180,E1 19927.018,E2 19927.018} C_VEL
LIN {X 0,Y 417.724,Z 888.46,A -85,B 0,C 180,E1 19924.722,E2 19924.722} C_VEL
LIN {X 0,Y 414.135,Z 903.782,A -85,B 0,C 180,E1 19922.406,E2 19922.406} C_VEL
LIN {X 0,Y 410.47,Z 919.761,A -85,B 0,C 180,E1 19919.586,E2 19919.586} C_VEL
LIN {X 0,Y 407.545,Z 933.141,A -85,B 0,C 180,E1 19916.831,E2 19916.831} C_VEL
LIN {X 0,Y 405.049,Z 945.262,A -85,B 0,C 180,E1 19913.877,E2 19913.877} C_VEL
LIN {X 0,Y 403.098,Z 956.149,A -85,B 0,C 180,E1 19910.772,E2 19910.772} C_VEL
LIN {X 0,Y 401.703,Z 965.1,A -85,B 0,C 180,E1 19907.675,E2 19907.675} C_VEL
LIN {X 0,Y 400.731,Z 973.109,A -85,B 0,C 180,E1 19904.299,E2 19904.299} C_VEL
LIN {X 0,Y 400.257,Z 978.565,A -85,B 0,C 180,E1 19901.38,E2 19901.38} C_VEL
LIN {X 0,Y 400.017,Z 983.277,A -85,B 0,C 180,E1 19898.045,E2 19898.045} C_VEL
LIN {X 0,Y 399.922,Z 986.001,A -85,B 0,C 180,E1 19895.163,E2 19895.163} C_VEL
LIN {X 0,Y 399.908,Z 987.712,A -85,B 0,C 180,E1 19892.005,E2 19892.005} C_VEL
LIN {X 0,Y 399.889,Z 987.879,A -85,B 0,C 180,E1 19888.997,E2 19888.997} C_VEL
LIN {X 0,Y 399.906,Z 986.923,A -85,B 0,C 180,E1 19886.129,E2 19886.129} C_VEL
LIN {X 0,Y 399.943,Z 984.304,A -85,B 0,C 180,E1 19882.82,E2 19882.82} C_VEL
LIN {X 0,Y 400.097,Z 980.937,A -85,B 0,C 180,E1 19880.071,E2 19880.071} C_VEL
LIN {X 0,Y 400.536,Z 975.353,A -85,B 0,C 180,E1 19876.724,E2 19876.724} C_VEL
LIN {X 0,Y 401.207,Z 969.02,A -85,B 0,C 180,E1 19873.794,E2 19873.794} C_VEL
LIN {X 0,Y 402.466,Z 959.992,A -85,B 0,C 180,E1 19870.406,E2 19870.406} C_VEL
LIN {X 0,Y 404.086,Z 950.461,A -85,B 0,C 180,E1 19867.45,E2 19867.45} C_VEL
LIN {X 0,Y 406.392,Z 938.538,A -85,B 0,C 180,E1 19864.343,E2 19864.343} C_VEL
LIN {X 0,Y 409.109,Z 925.97,A -85,B 0,C 180,E1 19861.541,E2 19861.541} C_VEL
LIN {X 0,Y 412.247,Z 911.949,A -85,B 0,C 180,E1 19858.889,E2 19858.889} C_VEL
LIN {X 0,Y 415.86,Z 896.486,A -85,B 0,C 180,E1 19856.349,E2 19856.349} C_VEL
LIN {X 0,Y 419.55,Z 880.475,A -85,B 0,C 180,E1 19854.112,E2 19854.112} C_VEL
LIN {X 0,Y 423.731,Z 862.147,A -85,B 0,C 180,E1 19851.904,E2 19851.904} C_VEL
LIN {X 0,Y 427.526,Z 844.479,A -85,B 0,C 180,E1 19850.094,E2 19850.094} C_VEL
LIN {X 0,Y 431.776,Z 823.363,A -85,B 0,C 180,E1 19848.265,E2 19848.265} C_VEL
LIN {X 0,Y 435.223,Z 804.55,A -85,B 0,C 180,E1 19846.9,E2 19846.9} C_VEL
LIN {X 0,Y 438.702,Z 782.928,A -85,B 0,C 180,E1 19845.604,E2 19845.604} C_VEL
LIN {X 0,Y 441.357,Z 763.698,A -85,B 0,C 180,E1 19844.662,E2 19844.662} C_VEL
LIN {X 0,Y 443.966,Z 740.239,A -85,B 0,C 180,E1 19843.762,E2 19843.762} C_VEL
LIN {X 0,Y 445.748,Z 719.358,A -85,B 0,C 180,E1 19843.169,E2 19843.169} C_VEL
LIN {X 0,Y 447.301,Z 686.453,A -85,B 0,C 180,E1 19842.519,E2 19842.519} C_VEL
LIN {X 0,Y 455.552,Z 472.833,A -85,B 0,C 180,E1 19838.607,E2 19838.607} C_VEL
LIN {X 0,Y 456.272,Z 452.391,A -85,B 0,C 180,E1 19838.212,E2 19838.212} C_VEL
LIN {X 0,Y 445.108,Z 436.21,A -85,B 0,C 180,E1 19835.895,E2 19835.895} C_VEL
LIN {X 0,Y 434.163,Z 421.491,A -85,B 0,C 180,E1 19833.395,E2 19833.395} C_VEL
LIN {X 0,Y 425.707,Z 410.818,A -85,B 0,C 180,E1 19831.27,E2 19831.27} C_VEL
LIN {X 0,Y 422.02,Z 406.045,A -85,B 0,C 180,E1 19830.269,E2 19830.269} C_VEL
LIN {X 0,Y 418.066,Z 401.6,A -85,B 0,C 180,E1 19829.163,E2 19829.163} C_VEL
LIN {X 0,Y 416.71,Z 399.685,A -85,B 0,C 180,E1 19828.756,E2 19828.756} C_VEL
LIN {X 0,Y 413.434,Z 396.304,A -85,B 0,C 180,E1 19827.785,E2 19827.785} C_VEL
LIN {X 0,Y 411.766,Z 393.736,A -85,B 0,C 180,E1 19827.24,E2 19827.24} C_VEL
LIN {X 0,Y 408.608,Z 391,A -85,B 0,C 180,E1 19826.251,E2 19826.251} C_VEL
LIN {X 0,Y 406.809,Z 387.58,A -85,B 0,C 180,E1 19825.589,E2 19825.589} C_VEL
LIN {X 0,Y 403.588,Z 385.505,A -85,B 0,C 180,E1 19824.518,E2 19824.518} C_VEL
LIN {X 0,Y 401.878,Z 382.653,A -85,B 0,C 180,E1 19823.847,E2 19823.847} C_VEL
LIN {X 0,Y 401.498,Z 380.977,A -85,B 0,C 180,E1 19823.604,E2 19823.604} C_VEL
LIN {X 0,Y 401.492,Z 381.024,A -85,B 0,C 180,E1 19819.646,E2 19819.646} C_VEL
LIN {X 0,Y 401.47,Z 380.988,A -85,B 0,C 180,E1 19815.752,E2 19815.752} C_VEL
LIN {X 0,Y 401.453,Z 381.026,A -85,B 0,C 180,E1 19811.93,E2 19811.93} C_VEL
LIN {X 0,Y 401.443,Z 381.027,A -85,B 0,C 180,E1 19808.018,E2 19808.018} C_VEL
LIN {X 0,Y 401.438,Z 381.03,A -85,B 0,C 180,E1 19804.142,E2 19804.142} C_VEL
LIN {X 0,Y 401.439,Z 381.032,A -85,B 0,C 180,E1 19800.286,E2 19800.286} C_VEL
LIN {X 0,Y 401.458,Z 381.03,A -85,B 0,C 180,E1 19796.574,E2 19796.574} C_VEL
LIN {X 0,Y 401.482,Z 381.031,A -85,B 0,C 180,E1 19792.703,E2 19792.703} C_VEL
LIN {X 0,Y 401.472,Z 381.04,A -85,B 0,C 180,E1 19788.654,E2 19788.654} C_VEL
LIN {X 0,Y 401.473,Z 381.028,A -85,B 0,C 180,E1 19784.693,E2 19784.693} C_VEL
LIN {X 0,Y 401.455,Z 381.001,A -85,B 0,C 180,E1 19780.807,E2 19780.807} C_VEL
LIN {X 0,Y 401.438,Z 380.996,A -85,B 0,C 180,E1 19777.059,E2 19777.059} C_VEL
LIN {X 0,Y 401.831,Z 382.579,A -85,B 0,C 180,E1 19776.654,E2 19776.654} C_VEL
LIN {X 0,Y 403.624,Z 385.536,A -85,B 0,C 180,E1 19775.953,E2 19775.953} C_VEL
LIN {X 0,Y 406.512,Z 387.813,A -85,B 0,C 180,E1 19774.973,E2 19774.973} C_VEL
LIN {X 0,Y 409.922,Z 392.464,A -85,B 0,C 180,E1 19773.802,E2 19773.802} C_VEL
LIN {X 0,Y 411.535,Z 394.14,A -85,B 0,C 180,E1 19773.291,E2 19773.291} C_VEL
LIN {X 0,Y 415.921,Z 399.636,A -85,B 0,C 180,E1 19771.929,E2 19771.929} C_VEL
LIN {X 0,Y 420.489,Z 405.584,A -85,B 0,C 180,E1 19770.592,E2 19770.592} C_VEL
LIN {X 0,Y 428.214,Z 415.793,A -85,B 0,C 180,E1 19768.504,E2 19768.504} C_VEL
LIN {X 0,Y 438.439,Z 430.168,A -85,B 0,C 180,E1 19765.994,E2 19765.994} C_VEL
LIN {X 0,Y 449.332,Z 446.653,A -85,B 0,C 180,E1 19763.57,E2 19763.57} C_VEL
LIN {X 0,Y 456.493,Z 458.459,A -85,B 0,C 180,E1 19762.084,E2 19762.084} C_VEL
LIN {X 0,Y 448.581,Z 663.35,A -85,B 0,C 180,E1 19758.323,E2 19758.323} C_VEL
LIN {X 0,Y 445.649,Z 738.115,A -85,B 0,C 180,E1 19756.937,E2 19756.937} C_VEL
LIN {X 0,Y 443.617,Z 761.463,A -85,B 0,C 180,E1 19756.32,E2 19756.32} C_VEL
LIN {X 0,Y 441.105,Z 783.99,A -85,B 0,C 180,E1 19755.51,E2 19755.51} C_VEL
LIN {X 0,Y 438.048,Z 805.777,A -85,B 0,C 180,E1 19754.48,E2 19754.48} C_VEL
LIN {X 0,Y 434.415,Z 828.447,A -85,B 0,C 180,E1 19753.147,E2 19753.147} C_VEL
LIN {X 0,Y 431.034,Z 847.041,A -85,B 0,C 180,E1 19751.823,E2 19751.823} C_VEL
LIN {X 0,Y 426.974,Z 867.682,A -85,B 0,C 180,E1 19750.084,E2 19750.084} C_VEL
LIN {X 0,Y 423.099,Z 886.1,A -85,B 0,C 180,E1 19748.25,E2 19748.25} C_VEL
LIN {X 0,Y 418.919,Z 905.368,A -85,B 0,C 180,E1 19745.992,E2 19745.992} C_VEL
LIN {X 0,Y 415.121,Z 922.664,A -85,B 0,C 180,E1 19743.636,E2 19743.636} C_VEL
LIN {X 0,Y 411.704,Z 938.22,A -85,B 0,C 180,E1 19741.147,E2 19741.147} C_VEL
LIN {X 0,Y 408.668,Z 952.733,A -85,B 0,C 180,E1 19738.492,E2 19738.492} C_VEL
LIN {X 0,Y 406.07,Z 965.82,A -85,B 0,C 180,E1 19735.678,E2 19735.678} C_VEL
LIN {X 0,Y 403.867,Z 978.294,A -85,B 0,C 180,E1 19732.563,E2 19732.563} C_VEL
LIN {X 0,Y 402.325,Z 988.291,A -85,B 0,C 180,E1 19729.601,E2 19729.601} C_VEL
LIN {X 0,Y 401.137,Z 997.808,A -85,B 0,C 180,E1 19726.209,E2 19726.209} C_VEL
LIN {X 0,Y 400.482,Z 1004.716,A -85,B 0,C 180,E1 19723.175,E2 19723.175} C_VEL
LIN {X 0,Y 400.085,Z 1010.433,A -85,B 0,C 180,E1 19719.929,E2 19719.929} C_VEL
LIN {X 0,Y 399.941,Z 1014.016,A -85,B 0,C 180,E1 19717.18,E2 19717.18} C_VEL
LIN {X 0,Y 399.911,Z 1016.767,A -85,B 0,C 180,E1 19713.993,E2 19713.993} C_VEL
LIN {X 0,Y 399.898,Z 1017.824,A -85,B 0,C 180,E1 19711.146,E2 19711.146} C_VEL
LIN {X 0,Y 399.906,Z 1017.733,A -85,B 0,C 180,E1 19708.281,E2 19708.281} C_VEL
LIN {X 0,Y 399.913,Z 1016.141,A -85,B 0,C 180,E1 19705.125,E2 19705.125} C_VEL
LIN {X 0,Y 399.962,Z 1013.524,A -85,B 0,C 180,E1 19702.388,E2 19702.388} C_VEL
LIN {X 0,Y 400.16,Z 1009.365,A -85,B 0,C 180,E1 19699.346,E2 19699.346} C_VEL
LIN {X 0,Y 400.569,Z 1003.566,A -85,B 0,C 180,E1 19696.285,E2 19696.285} C_VEL
LIN {X 0,Y 401.298,Z 996.358,A -85,B 0,C 180,E1 19693.203,E2 19693.203} C_VEL
LIN {X 0,Y 402.447,Z 987.357,A -85,B 0,C 180,E1 19690.103,E2 19690.103} C_VEL
LIN {X 0,Y 404.151,Z 976.619,A -85,B 0,C 180,E1 19686.971,E2 19686.971} C_VEL
LIN {X 0,Y 406.314,Z 964.532,A -85,B 0,C 180,E1 19684.026,E2 19684.026} C_VEL
LIN {X 0,Y 409.174,Z 950.19,A -85,B 0,C 180,E1 19681.021,E2 19681.021} C_VEL
LIN {X 0,Y 412.256,Z 935.647,A -85,B 0,C 180,E1 19678.412,E2 19678.412} C_VEL
LIN {X 0,Y 416.002,Z 918.557,A -85,B 0,C 180,E1 19675.782,E2 19675.782} C_VEL
LIN {X 0,Y 419.87,Z 901.142,A -85,B 0,C 180,E1 19673.469,E2 19673.469} C_VEL
LIN {X 0,Y 423.814,Z 882.716,A -85,B 0,C 180,E1 19671.396,E2 19671.396} C_VEL
LIN {X 0,Y 427.928,Z 863.066,A -85,B 0,C 180,E1 19669.498,E2 19669.498} C_VEL
LIN {X 0,Y 431.703,Z 843.397,A -85,B 0,C 180,E1 19667.9,E2 19667.9} C_VEL
LIN {X 0,Y 435.601,Z 821.225,A -85,B 0,C 180,E1 19666.396,E2 19666.396} C_VEL
LIN {X 0,Y 438.818,Z 800.578,A -85,B 0,C 180,E1 19665.253,E2 19665.253} C_VEL
LIN {X 0,Y 441.85,Z 777.663,A -85,B 0,C 180,E1 19664.248,E2 19664.248} C_VEL
LIN {X 0,Y 444.101,Z 756.825,A -85,B 0,C 180,E1 19663.542,E2 19663.542} C_VEL
LIN {X 0,Y 445.894,Z 733.091,A -85,B 0,C 180,E1 19662.964,E2 19662.964} C_VEL
LIN {X 0,Y 453.515,Z 532.626,A -85,B 0,C 180,E1 19659.286,E2 19659.286} C_VEL
LIN {X 0,Y 456.374,Z 458.035,A -85,B 0,C 180,E1 19657.894,E2 19657.894} C_VEL
LIN {X 0,Y 446.021,Z 441.548,A -85,B 0,C 180,E1 19655.73,E2 19655.73} C_VEL
LIN {X 0,Y 436.552,Z 427.556,A -85,B 0,C 180,E1 19653.581,E2 19653.581} C_VEL
LIN {X 0,Y 427.127,Z 414.268,A -85,B 0,C 180,E1 19651.232,E2 19651.232} C_VEL
LIN {X 0,Y 418.698,Z 403.218,A -85,B 0,C 180,E1 19648.919,E2 19648.919} C_VEL
LIN {X 0,Y 414.291,Z 397.578,A -85,B 0,C 180,E1 19647.605,E2 19647.605} C_VEL
LIN {X 0,Y 410.447,Z 392.908,A -85,B 0,C 180,E1 19646.396,E2 19646.396} C_VEL
LIN {X 0,Y 407.81,Z 389.761,A -85,B 0,C 180,E1 19645.524,E2 19645.524} C_VEL
LIN {X 0,Y 406.041,Z 387.276,A -85,B 0,C 180,E1 19644.902,E2 19644.902} C_VEL
LIN {X 0,Y 403.164,Z 384.989,A -85,B 0,C 180,E1 19643.921,E2 19643.921} C_VEL
LIN {X 0,Y 401.482,Z 381.235,A -85,B 0,C 180,E1 19643.105,E2 19643.105} C_VEL
LIN {X 0,Y 401.481,Z 381.004,A -85,B 0,C 180,E1 19639.494,E2 19639.494} C_VEL
LIN {X 0,Y 401.485,Z 381.008,A -85,B 0,C 180,E1 19635.454,E2 19635.454} C_VEL
LIN {X 0,Y 401.47,Z 381.032,A -85,B 0,C 180,E1 19631.492,E2 19631.492} C_VEL
LIN {X 0,Y 401.45,Z 381.041,A -85,B 0,C 180,E1 19627.585,E2 19627.585} C_VEL
LIN {X 0,Y 401.437,Z 381.044,A -85,B 0,C 180,E1 19623.713,E2 19623.713} C_VEL
LIN {X 0,Y 401.431,Z 381.045,A -85,B 0,C 180,E1 19619.857,E2 19619.857} C_VEL
LIN {X 0,Y 401.434,Z 381.041,A -85,B 0,C 180,E1 19616.001,E2 19616.001} C_VEL
LIN {X 0,Y 401.444,Z 381.035,A -85,B 0,C 180,E1 19612.126,E2 19612.126} C_VEL
LIN {X 0,Y 401.467,Z 381.028,A -85,B 0,C 180,E1 19608.361,E2 19608.361} C_VEL
LIN {X 0,Y 401.491,Z 381.005,A -85,B 0,C 180,E1 19604.504,E2 19604.504} C_VEL
LIN {X 0,Y 401.493,Z 381.005,A -85,B 0,C 180,E1 19600.506,E2 19600.506} C_VEL
LIN {X 0,Y 401.483,Z 380.982,A -85,B 0,C 180,E1 19596.673,E2 19596.673} C_VEL
LIN {X 0,Y 401.506,Z 381.122,A -85,B 0,C 180,E1 19596.207,E2 19596.207} C_VEL
LIN {X 0,Y 402.403,Z 383.877,A -85,B 0,C 180,E1 19595.796,E2 19595.796} C_VEL
LIN {X 0,Y 404.786,Z 386.54,A -85,B 0,C 180,E1 19594.936,E2 19594.936} C_VEL
LIN {X 0,Y 406.918,Z 387.892,A -85,B 0,C 180,E1 19594.239,E2 19594.239} C_VEL
LIN {X 0,Y 408.975,Z 391.47,A -85,B 0,C 180,E1 19593.501,E2 19593.501} C_VEL
LIN {X 0,Y 412.261,Z 394.307,A -85,B 0,C 180,E1 19592.482,E2 19592.482} C_VEL
LIN {X 0,Y 414.971,Z 398.207,A -85,B 0,C 180,E1 19591.623,E2 19591.623} C_VEL
LIN {X 0,Y 417.349,Z 400.439,A -85,B 0,C 180,E1 19590.939,E2 19590.939} C_VEL
LIN {X 0,Y 420.671,Z 404.788,A -85,B 0,C 180,E1 19589.979,E2 19589.979} C_VEL
LIN {X 0,Y 422.456,Z 406.802,A -85,B 0,C 180,E1 19589.491,E2 19589.491} C_VEL
LIN {X 0,Y 426.315,Z 411.404,A -85,B 0,C 180,E1 19588.465,E2 19588.465} C_VEL
LIN {X 0,Y 435.643,Z 423.58,A -85,B 0,C 180,E1 19586.141,E2 19586.141} C_VEL
LIN {X 0,Y 443.875,Z 434.632,A -85,B 0,C 180,E1 19584.269,E2 19584.269} C_VEL
LIN {X 0,Y 454.727,Z 450.043,A -85,B 0,C 180,E1 19581.999,E2 19581.999} C_VEL
LIN {X 0,Y 456.321,Z 452.769,A -85,B 0,C 180,E1 19581.673,E2 19581.673} C_VEL
LIN {X 0,Y 448.222,Z 661.009,A -85,B 0,C 180,E1 19577.852,E2 19577.852} C_VEL
LIN {X 0,Y 445.943,Z 716.568,A -85,B 0,C 180,E1 19576.81,E2 19576.81} C_VEL
LIN {X 0,Y 444.053,Z 739.079,A -85,B 0,C 180,E1 19576.184,E2 19576.184} C_VEL
LIN {X 0,Y 441.64,Z 761.485,A -85,B 0,C 180,E1 19575.346,E2 19575.346} C_VEL
LIN {X 0,Y 438.876,Z 781.638,A -85,B 0,C 180,E1 19574.373,E2 19574.373} C_VEL
LIN {X 0,Y 435.609,Z 802.44,A -85,B 0,C 180,E1 19573.151,E2 19573.151} C_VEL
LIN {X 0,Y 432.113,Z 821.553,A -85,B 0,C 180,E1 19571.783,E2 19571.783} C_VEL
LIN {X 0,Y 429.779,Z 833.515,A -85,B 0,C 180,E1 19570.804,E2 19570.804} C_VEL
LIN {X 0,Y 427.694,Z 840.189,A -85,B 0,C 180,E1 19570.314,E2 19570.314} C_VEL
LIN {X 0,Y 419.373,Z 856.657,A -85,B 0,C 180,E1 19569.239,E2 19569.239} C_VEL
LIN {X 0,Y 417.234,Z 862.725,A -85,B 0,C 180,E1 19568.669,E2 19568.669} C_VEL
LIN {X 0,Y 412.986,Z 880.47,A -85,B 0,C 180,E1 19566.506,E2 19566.506} C_VEL
LIN {X 0,Y 408.902,Z 897.253,A -85,B 0,C 180,E1 19564.132,E2 19564.132} C_VEL
LIN {X 0,Y 405.083,Z 912.687,A -85,B 0,C 180,E1 19561.548,E2 19561.548} C_VEL
LIN {X 0,Y 401.596,Z 927.273,A -85,B 0,C 180,E1 19558.715,E2 19558.715} C_VEL
LIN {X 0,Y 398.888,Z 939.121,A -85,B 0,C 180,E1 19556.015,E2 19556.015} C_VEL
LIN {X 0,Y 396.326,Z 951.492,A -85,B 0,C 180,E1 19552.702,E2 19552.702} C_VEL
LIN {X 0,Y 394.621,Z 960.937,A -85,B 0,C 180,E1 19549.69,E2 19549.69} C_VEL
LIN {X 0,Y 393.332,Z 969.464,A -85,B 0,C 180,E1 19546.387,E2 19546.387} C_VEL
LIN {X 0,Y 392.55,Z 976.365,A -85,B 0,C 180,E1 19543.1,E2 19543.1} C_VEL
LIN {X 0,Y 392.115,Z 981.519,A -85,B 0,C 180,E1 19539.835,E2 19539.835} C_VEL
LIN {X 0,Y 391.958,Z 984.975,A -85,B 0,C 180,E1 19536.885,E2 19536.885} C_VEL
LIN {X 0,Y 391.908,Z 987.314,A -85,B 0,C 180,E1 19533.656,E2 19533.656} C_VEL
LIN {X 0,Y 391.897,Z 988.187,A -85,B 0,C 180,E1 19530.877,E2 19530.877} C_VEL
LIN {X 0,Y 391.917,Z 987.949,A -85,B 0,C 180,E1 19527.66,E2 19527.66} C_VEL
LIN {X 0,Y 391.932,Z 986.26,A -85,B 0,C 180,E1 19524.584,E2 19524.584} C_VEL
LIN {X 0,Y 392.045,Z 983.366,A -85,B 0,C 180,E1 19521.494,E2 19521.494} C_VEL
LIN {X 0,Y 392.31,Z 978.771,A -85,B 0,C 180,E1 19518.236,E2 19518.236} C_VEL
LIN {X 0,Y 392.849,Z 973.298,A -85,B 0,C 180,E1 19515.256,E2 19515.256} C_VEL
LIN {X 0,Y 393.863,Z 965.642,A -85,B 0,C 180,E1 19511.96,E2 19511.96} C_VEL
LIN {X 0,Y 395.267,Z 957.162,A -85,B 0,C 180,E1 19508.951,E2 19508.951} C_VEL
LIN {X 0,Y 397.325,Z 946.449,A -85,B 0,C 180,E1 19505.786,E2 19505.786} C_VEL
LIN {X 0,Y 399.948,Z 934.49,A -85,B 0,C 180,E1 19502.777,E2 19502.777} C_VEL
LIN {X 0,Y 403.062,Z 921.031,A -85,B 0,C 180,E1 19499.931,E2 19499.931} C_VEL
LIN {X 0,Y 406.674,Z 906.25,A -85,B 0,C 180,E1 19497.23,E2 19497.23} C_VEL
LIN {X 0,Y 410.424,Z 890.964,A -85,B 0,C 180,E1 19494.852,E2 19494.852} C_VEL
LIN {X 0,Y 414.822,Z 872.844,A -85,B 0,C 180,E1 19492.429,E2 19492.429} C_VEL
LIN {X 0,Y 418.831,Z 855.786,A -85,B 0,C 180,E1 19490.487,E2 19490.487} C_VEL
LIN {X 0,Y 423.179,Z 836.133,A -85,B 0,C 180,E1 19488.586,E2 19488.586} C_VEL
LIN {X 0,Y 426.8,Z 818.396,A -85,B 0,C 180,E1 19487.128,E2 19487.128} C_VEL
LIN {X 0,Y 430.752,Z 796.707,A -85,B 0,C 180,E1 19485.638,E2 19485.638} C_VEL
LIN {X 0,Y 433.936,Z 776.842,A -85,B 0,C 180,E1 19484.515,E2 19484.515} C_VEL
LIN {X 0,Y 436.944,Z 754.066,A -85,B 0,C 180,E1 19483.493,E2 19483.493} C_VEL
LIN {X 0,Y 439.388,Z 731.255,A -85,B 0,C 180,E1 19482.711,E2 19482.711} C_VEL
LIN {X 0,Y 440.994,Z 708.429,A -85,B 0,C 180,E1 19482.165,E2 19482.165} C_VEL
LIN {X 0,Y 449.393,Z 501.376,A -85,B 0,C 180,E1 19478.334,E2 19478.334} C_VEL
LIN {X 0,Y 451.175,Z 456.347,A -85,B 0,C 180,E1 19477.477,E2 19477.477} C_VEL
LIN {X 0,Y 440.575,Z 441.095,A -85,B 0,C 180,E1 19475.201,E2 19475.201} C_VEL
LIN {X 0,Y 431.037,Z 428.098,A -85,B 0,C 180,E1 19472.954,E2 19472.954} C_VEL
LIN {X 0,Y 422.815,Z 417.612,A -85,B 0,C 180,E1 19470.835,E2 19470.835} C_VEL
LIN {X 0,Y 418.399,Z 412.137,A -85,B 0,C 180,E1 19469.609,E2 19469.609} C_VEL
LIN {X 0,Y 414.797,Z 407.505,A -85,B 0,C 180,E1 19468.547,E2 19468.547} C_VEL
LIN {X 0,Y 410.751,Z 403.036,A -85,B 0,C 180,E1 19467.313,E2 19467.313} C_VEL
LIN {X 0,Y 409.388,Z 401.047,A -85,B 0,C 180,E1 19466.861,E2 19466.861} C_VEL
LIN {X 0,Y 406.108,Z 397.888,A -85,B 0,C 180,E1 19465.796,E2 19465.796} C_VEL
LIN {X 0,Y 404.204,Z 394.9,A -85,B 0,C 180,E1 19465.102,E2 19465.102} C_VEL
LIN {X 0,Y 401.003,Z 392.235,A -85,B 0,C 180,E1 19463.981,E2 19463.981} C_VEL
LIN {X 0,Y 399.036,Z 388.599,A -85,B 0,C 180,E1 19463.166,E2 19463.166} C_VEL
LIN {X 0,Y 395.837,Z 386.673,A -85,B 0,C 180,E1 19461.953,E2 19461.953} C_VEL
LIN {X 0,Y 393.984,Z 383.816,A -85,B 0,C 180,E1 19461.123,E2 19461.123} C_VEL
LIN {X 0,Y 393.527,Z 382.019,A -85,B 0,C 180,E1 19460.837,E2 19460.837} C_VEL
LIN {X 0,Y 393.53,Z 381.962,A -85,B 0,C 180,E1 19456.989,E2 19456.989} C_VEL
LIN {X 0,Y 393.547,Z 382.021,A -85,B 0,C 180,E1 19453.069,E2 19453.069} C_VEL
LIN {X 0,Y 393.547,Z 382.014,A -85,B 0,C 180,E1 19449.063,E2 19449.063} C_VEL
LIN {X 0,Y 393.546,Z 382.012,A -85,B 0,C 180,E1 19445.102,E2 19445.102} C_VEL
LIN {X 0,Y 393.545,Z 382.01,A -85,B 0,C 180,E1 19441.019,E2 19441.019} C_VEL
LIN {X 0,Y 393.524,Z 382.013,A -85,B 0,C 180,E1 19437.088,E2 19437.088} C_VEL
LIN {X 0,Y 393.507,Z 382.018,A -85,B 0,C 180,E1 19433.142,E2 19433.142} C_VEL
LIN {X 0,Y 393.493,Z 382.027,A -85,B 0,C 180,E1 19429.311,E2 19429.311} C_VEL
LIN {X 0,Y 393.492,Z 382.035,A -85,B 0,C 180,E1 19425.431,E2 19425.431} C_VEL
LIN {X 0,Y 393.492,Z 381.98,A -85,B 0,C 180,E1 19421.385,E2 19421.385} C_VEL
LIN {X 0,Y 393.534,Z 382.259,A -85,B 0,C 180,E1 19419.611,E2 19419.611} C_VEL
LIN {X 0,Y 394.507,Z 385.033,A -85,B 0,C 180,E1 19419.101,E2 19419.101} C_VEL
LIN {X 0,Y 397.065,Z 387.692,A -85,B 0,C 180,E1 19418.042,E2 19418.042} C_VEL
LIN {X 0,Y 399.225,Z 388.973,A -85,B 0,C 180,E1 19417.236,E2 19417.236} C_VEL
LIN {X 0,Y 401.302,Z 392.587,A -85,B 0,C 180,E1 19416.39,E2 19416.39} C_VEL
LIN {X 0,Y 404.589,Z 395.551,A -85,B 0,C 180,E1 19415.236,E2 19415.236} C_VEL
LIN {X 0,Y 407.782,Z 399.826,A -85,B 0,C 180,E1 19414.123,E2 19414.123} C_VEL
LIN {X 0,Y 409.751,Z 402.154,A -85,B 0,C 180,E1 19413.478,E2 19413.478} C_VEL
LIN {X 0,Y 413.389,Z 406.684,A -85,B 0,C 180,E1 19412.33,E2 19412.33} C_VEL
LIN {X 0,Y 418.101,Z 412.943,A -85,B 0,C 180,E1 19410.919,E2 19410.919} C_VEL
LIN {X 0,Y 425.286,Z 422.523,A -85,B 0,C 180,E1 19408.933,E2 19408.933} C_VEL
LIN {X 0,Y 435.735,Z 437.446,A -85,B 0,C 180,E1 19406.308,E2 19406.308} C_VEL
LIN {X 0,Y 446.449,Z 453.988,A -85,B 0,C 180,E1 19403.874,E2 19403.874} C_VEL
LIN {X 0,Y 451.407,Z 462.396,A -85,B 0,C 180,E1 19402.812,E2 19402.812} C_VEL
LIN {X 0,Y 443.133,Z 666.584,A -85,B 0,C 180,E1 19399.036,E2 19399.036} C_VEL
LIN {X 0,Y 440.182,Z 738.046,A -85,B 0,C 180,E1 19397.697,E2 19397.697} C_VEL
LIN {X 0,Y 438.074,Z 761.302,A -85,B 0,C 180,E1 19397.078,E2 19397.078} C_VEL
LIN {X 0,Y 435.535,Z 783.223,A -85,B 0,C 180,E1 19396.291,E2 19396.291} C_VEL
LIN {X 0,Y 432.267,Z 805.478,A -85,B 0,C 180,E1 19395.238,E2 19395.238} C_VEL
LIN {X 0,Y 428.408,Z 828.461,A -85,B 0,C 180,E1 19393.875,E2 19393.875} C_VEL
LIN {X 0,Y 424.944,Z 846.665,A -85,B 0,C 180,E1 19392.57,E2 19392.57} C_VEL
LIN {X 0,Y 420.678,Z 867.375,A -85,B 0,C 180,E1 19390.809,E2 19390.809} C_VEL
LIN {X 0,Y 416.596,Z 885.795,A -85,B 0,C 180,E1 19388.957,E2 19388.957} C_VEL
LIN {X 0,Y 412.216,Z 904.91,A -85,B 0,C 180,E1 19386.694,E2 19386.694} C_VEL
LIN {X 0,Y 408.339,Z 921.609,A -85,B 0,C 180,E1 19384.394,E2 19384.394} C_VEL
LIN {X 0,Y 404.535,Z 937.905,A -85,B 0,C 180,E1 19381.763,E2 19381.763} C_VEL
LIN {X 0,Y 401.233,Z 952.753,A -85,B 0,C 180,E1 19378.994,E2 19378.994} C_VEL
LIN {X 0,Y 398.532,Z 965.506,A -85,B 0,C 180,E1 19376.201,E2 19376.201} C_VEL
LIN {X 0,Y 396.168,Z 977.981,A -85,B 0,C 180,E1 19373.026,E2 19373.026} C_VEL
LIN {X 0,Y 394.574,Z 987.509,A -85,B 0,C 180,E1 19370.157,E2 19370.157} C_VEL
LIN {X 0,Y 393.314,Z 996.773,A -85,B 0,C 180,E1 19366.845,E2 19366.845} C_VEL
LIN {X 0,Y 392.591,Z 1003.569,A -85,B 0,C 180,E1 19363.85,E2 19363.85} C_VEL
LIN {X 0,Y 392.149,Z 1009.49,A -85,B 0,C 180,E1 19360.577,E2 19360.577} C_VEL
LIN {X 0,Y 391.964,Z 1013.386,A -85,B 0,C 180,E1 19357.622,E2 19357.622} C_VEL
LIN {X 0,Y 391.913,Z 1016.074,A -85,B 0,C 180,E1 19354.683,E2 19354.683} C_VEL
LIN {X 0,Y 391.912,Z 1017.489,A -85,B 0,C 180,E1 19351.462,E2 19351.462} C_VEL
LIN {X 0,Y 391.909,Z 1017.513,A -85,B 0,C 180,E1 19348.685,E2 19348.685} C_VEL
LIN {X 0,Y 391.912,Z 1016.19,A -85,B 0,C 180,E1 19345.465,E2 19345.465} C_VEL
LIN {X 0,Y 391.955,Z 1013.55,A -85,B 0,C 180,E1 19342.526,E2 19342.526} C_VEL
LIN {X 0,Y 392.113,Z 1009.917,A -85,B 0,C 180,E1 19339.72,E2 19339.72} C_VEL
LIN {X 0,Y 392.567,Z 1003.882,A -85,B 0,C 180,E1 19336.3,E2 19336.3} C_VEL
LIN {X 0,Y 393.272,Z 997.137,A -85,B 0,C 180,E1 19333.306,E2 19333.306} C_VEL
LIN {X 0,Y 394.507,Z 987.985,A -85,B 0,C 180,E1 19329.995,E2 19329.995} C_VEL
LIN {X 0,Y 396.073,Z 978.517,A -85,B 0,C 180,E1 19327.126,E2 19327.126} C_VEL
LIN {X 0,Y 398.406,Z 966.161,A -85,B 0,C 180,E1 19323.952,E2 19323.952} C_VEL
LIN {X 0,Y 401.143,Z 953.138,A -85,B 0,C 180,E1 19321.087,E2 19321.087} C_VEL
LIN {X 0,Y 404.342,Z 938.77,A -85,B 0,C 180,E1 19318.388,E2 19318.388} C_VEL
LIN {X 0,Y 408.036,Z 922.931,A -85,B 0,C 180,E1 19315.799,E2 19315.799} C_VEL
LIN {X 0,Y 411.952,Z 906.036,A -85,B 0,C 180,E1 19313.453,E2 19313.453} C_VEL
LIN {X 0,Y 416.145,Z 887.86,A -85,B 0,C 180,E1 19311.265,E2 19311.265} C_VEL
LIN {X 0,Y 420.234,Z 869.301,A -85,B 0,C 180,E1 19309.375,E2 19309.375} C_VEL
LIN {X 0,Y 424.58,Z 848.534,A -85,B 0,C 180,E1 19307.577,E2 19307.577} C_VEL
LIN {X 0,Y 428.215,Z 829.451,A -85,B 0,C 180,E1 19306.193,E2 19306.193} C_VEL
LIN {X 0,Y 432.066,Z 806.729,A -85,B 0,C 180,E1 19304.831,E2 19304.831} C_VEL
LIN {X 0,Y 435.237,Z 785.127,A -85,B 0,C 180,E1 19303.794,E2 19303.794} C_VEL
LIN {X 0,Y 437.966,Z 762.136,A -85,B 0,C 180,E1 19302.949,E2 19302.949} C_VEL
LIN {X 0,Y 440.117,Z 738.849,A -85,B 0,C 180,E1 19302.321,E2 19302.321} C_VEL
LIN {X 0,Y 442.673,Z 677.858,A -85,B 0,C 180,E1 19301.173,E2 19301.173} C_VEL
LIN {X 0,Y 450.933,Z 472.833,A -85,B 0,C 180,E1 19297.386,E2 19297.386} C_VEL
LIN {X 0,Y 451.261,Z 461.896,A -85,B 0,C 180,E1 19297.16,E2 19297.16} C_VEL
LIN {X 0,Y 441.344,Z 446.052,A -85,B 0,C 180,E1 19295.011,E2 19295.011} C_VEL
LIN {X 0,Y 432.788,Z 433.251,A -85,B 0,C 180,E1 19293,E2 19293} C_VEL
LIN {X 0,Y 423.981,Z 420.737,A -85,B 0,C 180,E1 19290.74,E2 19290.74} C_VEL
LIN {X 0,Y 415.908,Z 410.005,A -85,B 0,C 180,E1 19288.463,E2 19288.463} C_VEL
LIN {X 0,Y 411.677,Z 404.511,A -85,B 0,C 180,E1 19287.168,E2 19287.168} C_VEL
LIN {X 0,Y 408.093,Z 400.108,A -85,B 0,C 180,E1 19286.012,E2 19286.012} C_VEL
LIN {X 0,Y 405.044,Z 396.232,A -85,B 0,C 180,E1 19284.968,E2 19284.968} C_VEL
LIN {X 0,Y 403.74,Z 394.656,A -85,B 0,C 180,E1 19284.507,E2 19284.507} C_VEL
LIN {X 0,Y 400.763,Z 391.889,A -85,B 0,C 180,E1 19283.449,E2 19283.449} C_VEL
LIN {X 0,Y 398.954,Z 388.595,A -85,B 0,C 180,E1 19282.703,E2 19282.703} C_VEL
LIN {X 0,Y 395.755,Z 386.596,A -85,B 0,C 180,E1 19281.489,E2 19281.489} C_VEL
LIN {X 0,Y 393.969,Z 383.898,A -85,B 0,C 180,E1 19280.695,E2 19280.695} C_VEL
LIN {X 0,Y 393.503,Z 382.025,A -85,B 0,C 180,E1 19280.367,E2 19280.367} C_VEL
LIN {X 0,Y 393.489,Z 381.978,A -85,B 0,C 180,E1 19276.382,E2 19276.382} C_VEL
LIN {X 0,Y 393.491,Z 382.018,A -85,B 0,C 180,E1 19272.473,E2 19272.473} C_VEL
LIN {X 0,Y 393.486,Z 382.021,A -85,B 0,C 180,E1 19268.475,E2 19268.475} C_VEL
LIN {X 0,Y 393.499,Z 382.022,A -85,B 0,C 180,E1 19264.664,E2 19264.664} C_VEL
LIN {X 0,Y 393.515,Z 382.025,A -85,B 0,C 180,E1 19260.728,E2 19260.728} C_VEL
LIN {X 0,Y 393.535,Z 382.026,A -85,B 0,C 180,E1 19256.86,E2 19256.86} C_VEL
LIN {X 0,Y 393.559,Z 382.026,A -85,B 0,C 180,E1 19252.849,E2 19252.849} C_VEL
LIN {X 0,Y 393.547,Z 382.019,A -85,B 0,C 180,E1 19248.718,E2 19248.718} C_VEL
LIN {X 0,Y 393.559,Z 381.995,A -85,B 0,C 180,E1 19244.679,E2 19244.679} C_VEL
LIN {X 0,Y 393.551,Z 381.989,A -85,B 0,C 180,E1 19240.56,E2 19240.56} C_VEL
LIN {X 0,Y 393.558,Z 382.226,A -85,B 0,C 180,E1 19238.973,E2 19238.973} C_VEL
LIN {X 0,Y 394.512,Z 384.908,A -85,B 0,C 180,E1 19238.478,E2 19238.478} C_VEL
LIN {X 0,Y 396.718,Z 387.448,A -85,B 0,C 180,E1 19237.553,E2 19237.553} C_VEL
LIN {X 0,Y 399.198,Z 388.899,A -85,B 0,C 180,E1 19236.629,E2 19236.629} C_VEL
LIN {X 0,Y 401.143,Z 392.421,A -85,B 0,C 180,E1 19235.833,E2 19235.833} C_VEL
LIN {X 0,Y 404.074,Z 394.827,A -85,B 0,C 180,E1 19234.811,E2 19234.811} C_VEL
LIN {X 0,Y 404.818,Z 395.752,A -85,B 0,C 180,E1 19234.547,E2 19234.547} C_VEL
LIN {X 0,Y 407.434,Z 399.474,A -85,B 0,C 180,E1 19233.629,E2 19233.629} C_VEL
LIN {X 0,Y 409.968,Z 401.777,A -85,B 0,C 180,E1 19232.827,E2 19232.827} C_VEL
LIN {X 0,Y 413.191,Z 405.987,A -85,B 0,C 180,E1 19231.805,E2 19231.805} C_VEL
LIN {X 0,Y 415.025,Z 407.922,A -85,B 0,C 180,E1 19231.261,E2 19231.261} C_VEL
LIN {X 0,Y 418.742,Z 412.466,A -85,B 0,C 180,E1 19230.181,E2 19230.181} C_VEL
LIN {X 0,Y 425.326,Z 420.862,A -85,B 0,C 180,E1 19228.383,E2 19228.383} C_VEL
LIN {X 0,Y 432.024,Z 429.446,A -85,B 0,C 180,E1 19226.696,E2 19226.696} C_VEL
LIN {X 0,Y 442.655,Z 443.969,A -85,B 0,C 180,E1 19224.235,E2 19224.235} C_VEL
LIN {X 0,Y 451.249,Z 456.72,A -85,B 0,C 180,E1 19222.402,E2 19222.402} C_VEL
LIN {X 0,Y 442.654,Z 667.552,A -85,B 0,C 180,E1 19218.505,E2 19218.505} C_VEL
LIN {X 0,Y 440.492,Z 717.07,A -85,B 0,C 180,E1 19217.565,E2 19217.565} C_VEL
LIN {X 0,Y 438.527,Z 739.525,A -85,B 0,C 180,E1 19216.936,E2 19216.936} C_VEL
LIN {X 0,Y 435.925,Z 762.533,A -85,B 0,C 180,E1 19216.064,E2 19216.064} C_VEL
LIN {X 0,Y 433.149,Z 781.95,A -85,B 0,C 180,E1 19215.119,E2 19215.119} C_VEL
LIN {X 0,Y 429.743,Z 802.752,A -85,B 0,C 180,E1 19213.888,E2 19213.888} C_VEL
LIN {X 0,Y 426.094,Z 821.864,A -85,B 0,C 180,E1 19212.511,E2 19212.511} C_VEL
LIN {X 0,Y 422.01,Z 841.611,A -85,B 0,C 180,E1 19210.832,E2 19210.832} C_VEL
LIN {X 0,Y 417.772,Z 860.27,A -85,B 0,C 180,E1 19208.938,E2 19208.938} C_VEL
LIN {X 0,Y 417.234,Z 862.725,A -85,B 0,C 180,E1 19208.669,E2 19208.669} C_VEL
LIN {X 0,Y 415.078,Z 868.798,A -85,B 0,C 180,E1 19208.072,E2 19208.072} C_VEL
LIN {X 0,Y 406.43,Z 884.023,A -85,B 0,C 180,E1 19206.685,E2 19206.685} C_VEL
LIN {X 0,Y 404.155,Z 889.548,A -85,B 0,C 180,E1 19205.986,E2 19205.986} C_VEL
LIN {X 0,Y 400.29,Z 904.41,A -85,B 0,C 180,E1 19203.673,E2 19203.673} C_VEL
LIN {X 0,Y 396.206,Z 920.177,A -85,B 0,C 180,E1 19200.812,E2 19200.812} C_VEL
LIN {X 0,Y 392.925,Z 933.439,A -85,B 0,C 180,E1 19197.994,E2 19197.994} C_VEL
LIN {X 0,Y 390.003,Z 945.889,A -85,B 0,C 180,E1 19194.859,E2 19194.859} C_VEL
LIN {X 0,Y 387.74,Z 956.773,A -85,B 0,C 180,E1 19191.636,E2 19191.636} C_VEL
LIN {X 0,Y 386.105,Z 965.72,A -85,B 0,C 180,E1 19188.414,E2 19188.414} C_VEL
LIN {X 0,Y 384.945,Z 973.725,A -85,B 0,C 180,E1 19184.898,E2 19184.898} C_VEL
LIN {X 0,Y 384.366,Z 979.176,A -85,B 0,C 180,E1 19181.857,E2 19181.857} C_VEL
LIN {X 0,Y 384.058,Z 983.884,A -85,B 0,C 180,E1 19178.382,E2 19178.382} C_VEL
LIN {X 0,Y 383.939,Z 986.604,A -85,B 0,C 180,E1 19175.378,E2 19175.378} C_VEL
LIN {X 0,Y 383.921,Z 988.312,A -85,B 0,C 180,E1 19172.089,E2 19172.089} C_VEL
LIN {X 0,Y 383.902,Z 988.478,A -85,B 0,C 180,E1 19168.955,E2 19168.955} C_VEL
LIN {X 0,Y 383.925,Z 987.523,A -85,B 0,C 180,E1 19165.968,E2 19165.968} C_VEL
LIN {X 0,Y 383.972,Z 985.061,A -85,B 0,C 180,E1 19162.67,E2 19162.67} C_VEL
LIN {X 0,Y 384.155,Z 981.742,A -85,B 0,C 180,E1 19159.806,E2 19159.806} C_VEL
LIN {X 0,Y 384.649,Z 976.514,A -85,B 0,C 180,E1 19156.453,E2 19156.453} C_VEL
LIN {X 0,Y 385.455,Z 969.973,A -85,B 0,C 180,E1 19153.267,E2 19153.267} C_VEL
LIN {X 0,Y 386.838,Z 961.501,A -85,B 0,C 180,E1 19149.896,E2 19149.896} C_VEL
LIN {X 0,Y 388.661,Z 952.08,A -85,B 0,C 180,E1 19146.824,E2 19146.824} C_VEL
LIN {X 0,Y 391.393,Z 939.773,A -85,B 0,C 180,E1 19143.448,E2 19143.448} C_VEL
LIN {X 0,Y 394.435,Z 927.271,A -85,B 0,C 180,E1 19140.546,E2 19140.546} C_VEL
LIN {X 0,Y 398.157,Z 912.611,A -85,B 0,C 180,E1 19137.667,E2 19137.667} C_VEL
LIN {X 0,Y 402.273,Z 896.895,A -85,B 0,C 180,E1 19135.016,E2 19135.016} C_VEL
LIN {X 0,Y 406.477,Z 880.535,A -85,B 0,C 180,E1 19132.679,E2 19132.679} C_VEL
LIN {X 0,Y 411.173,Z 861.734,A -85,B 0,C 180,E1 19130.379,E2 19130.379} C_VEL
LIN {X 0,Y 415.357,Z 844.118,A -85,B 0,C 180,E1 19128.554,E2 19128.554} C_VEL
LIN {X 0,Y 419.793,Z 823.956,A -85,B 0,C 180,E1 19126.788,E2 19126.788} C_VEL
LIN {X 0,Y 423.37,Z 806.039,A -85,B 0,C 180,E1 19125.465,E2 19125.465} C_VEL
LIN {X 0,Y 427.125,Z 784.79,A -85,B 0,C 180,E1 19124.159,E2 19124.159} C_VEL
LIN {X 0,Y 429.992,Z 765.75,A -85,B 0,C 180,E1 19123.205,E2 19123.205} C_VEL
LIN {X 0,Y 432.824,Z 742.885,A -85,B 0,C 180,E1 19122.298,E2 19122.298} C_VEL
LIN {X 0,Y 434.763,Z 722.164,A -85,B 0,C 180,E1 19121.688,E2 19121.688} C_VEL
LIN {X 0,Y 436.461,Z 691.434,A -85,B 0,C 180,E1 19121.053,E2 19121.053} C_VEL
LIN {X 0,Y 445.419,Z 480.365,A -85,B 0,C 180,E1 19117.128,E2 19117.128} C_VEL
LIN {X 0,Y 446.229,Z 460.588,A -85,B 0,C 180,E1 19116.746,E2 19116.746} C_VEL
LIN {X 0,Y 435.262,Z 444.623,A -85,B 0,C 180,E1 19114.29,E2 19114.29} C_VEL
LIN {X 0,Y 424.352,Z 429.923,A -85,B 0,C 180,E1 19111.579,E2 19111.579} C_VEL
LIN {X 0,Y 419.279,Z 423.63,A -85,B 0,C 180,E1 19110.21,E2 19110.21} C_VEL
LIN {X 0,Y 415.6,Z 418.956,A -85,B 0,C 180,E1 19109.156,E2 19109.156} C_VEL
LIN {X 0,Y 411.426,Z 413.73,A -85,B 0,C 180,E1 19107.893,E2 19107.893} C_VEL
LIN {X 0,Y 407.812,Z 409.31,A -85,B 0,C 180,E1 19106.737,E2 19106.737} C_VEL
LIN {X 0,Y 406.424,Z 407.842,A -85,B 0,C 180,E1 19106.284,E2 19106.284} C_VEL
LIN {X 0,Y 403.141,Z 404.013,A -85,B 0,C 180,E1 19105.155,E2 19105.155} C_VEL
LIN {X 0,Y 401.924,Z 402.258,A -85,B 0,C 180,E1 19104.704,E2 19104.704} C_VEL
LIN {X 0,Y 398.632,Z 399.146,A -85,B 0,C 180,E1 19103.504,E2 19103.504} C_VEL
LIN {X 0,Y 397.015,Z 396.221,A -85,B 0,C 180,E1 19102.82,E2 19102.82} C_VEL
LIN {X 0,Y 393.734,Z 393.867,A -85,B 0,C 180,E1 19101.528,E2 19101.528} C_VEL
LIN {X 0,Y 391.648,Z 390.383,A -85,B 0,C 180,E1 19100.551,E2 19100.551} C_VEL
LIN {X 0,Y 391.21,Z 389.69,A -85,B 0,C 180,E1 19100.34,E2 19100.34} C_VEL
LIN {X 0,Y 387.812,Z 387.589,A -85,B 0,C 180,E1 19098.801,E2 19098.801} C_VEL
LIN {X 0,Y 386.102,Z 384.944,A -85,B 0,C 180,E1 19097.871,E2 19097.871} C_VEL
LIN {X 0,Y 385.609,Z 382.948,A -85,B 0,C 180,E1 19097.505,E2 19097.505} C_VEL
LIN {X 0,Y 385.611,Z 383.016,A -85,B 0,C 180,E1 19093.495,E2 19093.495} C_VEL
LIN {X 0,Y 385.603,Z 383.007,A -85,B 0,C 180,E1 19089.402,E2 19089.402} C_VEL
LIN {X 0,Y 385.582,Z 383.006,A -85,B 0,C 180,E1 19085.506,E2 19085.506} C_VEL
LIN {X 0,Y 385.565,Z 383.006,A -85,B 0,C 180,E1 19081.635,E2 19081.635} C_VEL
LIN {X 0,Y 385.552,Z 383.005,A -85,B 0,C 180,E1 19077.771,E2 19077.771} C_VEL
LIN {X 0,Y 385.547,Z 383.005,A -85,B 0,C 180,E1 19073.747,E2 19073.747} C_VEL
LIN {X 0,Y 385.545,Z 383.011,A -85,B 0,C 180,E1 19069.692,E2 19069.692} C_VEL
LIN {X 0,Y 385.552,Z 383.024,A -85,B 0,C 180,E1 19065.585,E2 19065.585} C_VEL
LIN {X 0,Y 385.591,Z 383.148,A -85,B 0,C 180,E1 19062.962,E2 19062.962} C_VEL
LIN {X 0,Y 386.555,Z 385.886,A -85,B 0,C 180,E1 19062.346,E2 19062.346} C_VEL
LIN {X 0,Y 388.864,Z 388.505,A -85,B 0,C 180,E1 19061.175,E2 19061.175} C_VEL
LIN {X 0,Y 391.438,Z 389.934,A -85,B 0,C 180,E1 19060.039,E2 19060.039} C_VEL
LIN {X 0,Y 393.121,Z 393.195,A -85,B 0,C 180,E1 19059.219,E2 19059.219} C_VEL
LIN {X 0,Y 396.319,Z 395.912,A -85,B 0,C 180,E1 19057.92,E2 19057.92} C_VEL
LIN {X 0,Y 397.193,Z 396.629,A -85,B 0,C 180,E1 19057.582,E2 19057.582} C_VEL
LIN {X 0,Y 399.712,Z 400.449,A -85,B 0,C 180,E1 19056.564,E2 19056.564} C_VEL
LIN {X 0,Y 402.59,Z 403.101,A -85,B 0,C 180,E1 19055.536,E2 19055.536} C_VEL
LIN {X 0,Y 405.852,Z 407.373,A -85,B 0,C 180,E1 19054.383,E2 19054.383} C_VEL
LIN {X 0,Y 410.978,Z 413.87,A -85,B 0,C 180,E1 19052.704,E2 19052.704} C_VEL
LIN {X 0,Y 415.625,Z 420.128,A -85,B 0,C 180,E1 19051.28,E2 19051.28} C_VEL
LIN {X 0,Y 422.604,Z 429.583,A -85,B 0,C 180,E1 19049.306,E2 19049.306} C_VEL
LIN {X 0,Y 433.409,Z 445.223,A -85,B 0,C 180,E1 19046.54,E2 19046.54} C_VEL
LIN {X 0,Y 444.472,Z 462.719,A -85,B 0,C 180,E1 19043.987,E2 19043.987} C_VEL
LIN {X 0,Y 446.401,Z 466.208,A -85,B 0,C 180,E1 19043.559,E2 19043.559} C_VEL
LIN {X 0,Y 437.711,Z 670.897,A -85,B 0,C 180,E1 19039.746,E2 19039.746} C_VEL
LIN {X 0,Y 434.789,Z 738.084,A -85,B 0,C 180,E1 19038.475,E2 19038.475} C_VEL
LIN {X 0,Y 432.596,Z 761.273,A -85,B 0,C 180,E1 19037.852,E2 19037.852} C_VEL
LIN {X 0,Y 429.861,Z 783.686,A -85,B 0,C 180,E1 19037.038,E2 19037.038} C_VEL
LIN {X 0,Y 426.569,Z 805.179,A -85,B 0,C 180,E1 19036.015,E2 19036.015} C_VEL
LIN {X 0,Y 422.534,Z 828.159,A -85,B 0,C 180,E1 19034.646,E2 19034.646} C_VEL
LIN {X 0,Y 418.718,Z 847.34,A -85,B 0,C 180,E1 19033.256,E2 19033.256} C_VEL
LIN {X 0,Y 414.103,Z 868.553,A -85,B 0,C 180,E1 19031.415,E2 19031.415} C_VEL
LIN {X 0,Y 409.857,Z 886.833,A -85,B 0,C 180,E1 19029.542,E2 19029.542} C_VEL
LIN {X 0,Y 405.434,Z 905.021,A -85,B 0,C 180,E1 19027.345,E2 19027.345} C_VEL
LIN {X 0,Y 401.231,Z 922.249,A -85,B 0,C 180,E1 19024.93,E2 19024.93} C_VEL
LIN {X 0,Y 397.205,Z 938.475,A -85,B 0,C 180,E1 19022.244,E2 19022.244} C_VEL
LIN {X 0,Y 393.645,Z 953.532,A -85,B 0,C 180,E1 19019.352,E2 19019.352} C_VEL
LIN {X 0,Y 390.893,Z 965.839,A -85,B 0,C 180,E1 19016.589,E2 19016.589} C_VEL
LIN {X 0,Y 388.275,Z 978.808,A -85,B 0,C 180,E1 19013.174,E2 19013.174} C_VEL
LIN {X 0,Y 386.569,Z 988.607,A -85,B 0,C 180,E1 19010.119,E2 19010.119} C_VEL
LIN {X 0,Y 385.288,Z 997.552,A -85,B 0,C 180,E1 19006.74,E2 19006.74} C_VEL
LIN {X 0,Y 384.54,Z 1004.507,A -85,B 0,C 180,E1 19003.532,E2 19003.532} C_VEL
LIN {X 0,Y 384.104,Z 1010.037,A -85,B 0,C 180,E1 19000.195,E2 19000.195} C_VEL
LIN {X 0,Y 383.946,Z 1013.576,A -85,B 0,C 180,E1 18997.331,E2 18997.331} C_VEL
LIN {X 0,Y 383.92,Z 1016.226,A -85,B 0,C 180,E1 18994.032,E2 18994.032} C_VEL
LIN {X 0,Y 383.911,Z 1017.236,A -85,B 0,C 180,E1 18991.194,E2 18991.194} C_VEL
LIN {X 0,Y 383.917,Z 1017.165,A -85,B 0,C 180,E1 18988.359,E2 18988.359} C_VEL
LIN {X 0,Y 383.923,Z 1015.539,A -85,B 0,C 180,E1 18984.921,E2 18984.921} C_VEL
LIN {X 0,Y 384.009,Z 1012.755,A -85,B 0,C 180,E1 18981.919,E2 18981.919} C_VEL
LIN {X 0,Y 384.239,Z 1007.981,A -85,B 0,C 180,E1 18978.443,E2 18978.443} C_VEL
LIN {X 0,Y 384.73,Z 1002.328,A -85,B 0,C 180,E1 18975.401,E2 18975.401} C_VEL
LIN {X 0,Y 385.687,Z 994.544,A -85,B 0,C 180,E1 18972.034,E2 18972.034} C_VEL
LIN {X 0,Y 387.029,Z 985.795,A -85,B 0,C 180,E1 18968.958,E2 18968.958} C_VEL
LIN {X 0,Y 389.157,Z 974.321,A -85,B 0,C 180,E1 18965.569,E2 18965.569} C_VEL
LIN {X 0,Y 391.601,Z 962.607,A -85,B 0,C 180,E1 18962.643,E2 18962.643} C_VEL
LIN {X 0,Y 394.875,Z 948.219,A -85,B 0,C 180,E1 18959.579,E2 18959.579} C_VEL
LIN {X 0,Y 398.502,Z 933.296,A -85,B 0,C 180,E1 18956.845,E2 18956.845} C_VEL
LIN {X 0,Y 402.504,Z 916.896,A -85,B 0,C 180,E1 18954.29,E2 18954.29} C_VEL
LIN {X 0,Y 406.861,Z 899.3,A -85,B 0,C 180,E1 18951.921,E2 18951.921} C_VEL
LIN {X 0,Y 411.124,Z 881.412,A -85,B 0,C 180,E1 18949.879,E2 18949.879} C_VEL
LIN {X 0,Y 415.575,Z 861.954,A -85,B 0,C 180,E1 18947.973,E2 18947.973} C_VEL
LIN {X 0,Y 419.609,Z 842.862,A -85,B 0,C 180,E1 18946.4,E2 18946.4} C_VEL
LIN {X 0,Y 424.038,Z 819.91,A -85,B 0,C 180,E1 18944.831,E2 18944.831} C_VEL
LIN {X 0,Y 427.427,Z 799.955,A -85,B 0,C 180,E1 18943.719,E2 18943.719} C_VEL
LIN {X 0,Y 430.695,Z 777.191,A -85,B 0,C 180,E1 18942.711,E2 18942.711} C_VEL
LIN {X 0,Y 433.046,Z 757.142,A -85,B 0,C 180,E1 18942.025,E2 18942.025} C_VEL
LIN {X 0,Y 435.065,Z 732.73,A -85,B 0,C 180,E1 18941.418,E2 18941.418} C_VEL
LIN {X 0,Y 443.424,Z 533.409,A -85,B 0,C 180,E1 18937.701,E2 18937.701} C_VEL
LIN {X 0,Y 446.285,Z 465.768,A -85,B 0,C 180,E1 18936.42,E2 18936.42} C_VEL
LIN {X 0,Y 436.011,Z 449.368,A -85,B 0,C 180,E1 18934.103,E2 18934.103} C_VEL
LIN {X 0,Y 426.969,Z 435.942,A -85,B 0,C 180,E1 18931.874,E2 18931.874} C_VEL
LIN {X 0,Y 418.031,Z 423.202,A -85,B 0,C 180,E1 18929.44,E2 18929.44} C_VEL
LIN {X 0,Y 412.416,Z 415.895,A -85,B 0,C 180,E1 18927.78,E2 18927.78} C_VEL
LIN {X 0,Y 409.191,Z 411.545,A -85,B 0,C 180,E1 18926.757,E2 18926.757} C_VEL
LIN {X 0,Y 405.562,Z 407.1,A -85,B 0,C 180,E1 18925.558,E2 18925.558} C_VEL
LIN {X 0,Y 401.657,Z 402.101,A -85,B 0,C 180,E1 18924.173,E2 18924.173} C_VEL
LIN {X 0,Y 398.476,Z 398.904,A -85,B 0,C 180,E1 18923.004,E2 18923.004} C_VEL
LIN {X 0,Y 396.93,Z 396.193,A -85,B 0,C 180,E1 18922.356,E2 18922.356} C_VEL
LIN {X 0,Y 393.645,Z 393.8,A -85,B 0,C 180,E1 18921.064,E2 18921.064} C_VEL
LIN {X 0,Y 391.691,Z 390.635,A -85,B 0,C 180,E1 18920.158,E2 18920.158} C_VEL
LIN {X 0,Y 391.279,Z 389.686,A -85,B 0,C 180,E1 18919.946,E2 18919.946} C_VEL
LIN {X 0,Y 387.851,Z 387.644,A -85,B 0,C 180,E1 18918.409,E2 18918.409} C_VEL
LIN {X 0,Y 386.069,Z 384.839,A -85,B 0,C 180,E1 18917.444,E2 18917.444} C_VEL
LIN {X 0,Y 385.568,Z 382.954,A -85,B 0,C 180,E1 18917.039,E2 18917.039} C_VEL
LIN {X 0,Y 385.589,Z 383.005,A -85,B 0,C 180,E1 18913.19,E2 18913.19} C_VEL
LIN {X 0,Y 385.584,Z 383.003,A -85,B 0,C 180,E1 18909.101,E2 18909.101} C_VEL
LIN {X 0,Y 385.59,Z 383.002,A -85,B 0,C 180,E1 18905.207,E2 18905.207} C_VEL
LIN {X 0,Y 385.594,Z 383.004,A -85,B 0,C 180,E1 18901.188,E2 18901.188} C_VEL
LIN {X 0,Y 385.588,Z 383.01,A -85,B 0,C 180,E1 18897.176,E2 18897.176} C_VEL
LIN {X 0,Y 385.591,Z 383.017,A -85,B 0,C 180,E1 18893.149,E2 18893.149} C_VEL
LIN {X 0,Y 385.582,Z 383.02,A -85,B 0,C 180,E1 18889.239,E2 18889.239} C_VEL
LIN {X 0,Y 385.577,Z 383.008,A -85,B 0,C 180,E1 18885.278,E2 18885.278} C_VEL
LIN {X 0,Y 385.625,Z 383.148,A -85,B 0,C 180,E1 18882.294,E2 18882.294} C_VEL
LIN {X 0,Y 386.512,Z 385.852,A -85,B 0,C 180,E1 18881.72,E2 18881.72} C_VEL
LIN {X 0,Y 388.838,Z 388.453,A -85,B 0,C 180,E1 18880.549,E2 18880.549} C_VEL
LIN {X 0,Y 391.525,Z 390.065,A -85,B 0,C 180,E1 18879.364,E2 18879.364} C_VEL
LIN {X 0,Y 393.435,Z 393.54,A -85,B 0,C 180,E1 18878.455,E2 18878.455} C_VEL
LIN {X 0,Y 396.329,Z 395.897,A -85,B 0,C 180,E1 18877.295,E2 18877.295} C_VEL
LIN {X 0,Y 397.199,Z 396.69,A -85,B 0,C 180,E1 18876.956,E2 18876.956} C_VEL
LIN {X 0,Y 399.734,Z 400.486,A -85,B 0,C 180,E1 18875.938,E2 18875.938} C_VEL
LIN {X 0,Y 402.536,Z 402.993,A -85,B 0,C 180,E1 18874.944,E2 18874.944} C_VEL
LIN {X 0,Y 405.507,Z 407.031,A -85,B 0,C 180,E1 18873.888,E2 18873.888} C_VEL
LIN {X 0,Y 407.699,Z 409.162,A -85,B 0,C 180,E1 18873.176,E2 18873.176} C_VEL
LIN {X 0,Y 411.313,Z 413.642,A -85,B 0,C 180,E1 18872.02,E2 18872.02} C_VEL
LIN {X 0,Y 413.113,Z 415.925,A -85,B 0,C 180,E1 18871.466,E2 18871.466} C_VEL
LIN {X 0,Y 417.544,Z 421.398,A -85,B 0,C 180,E1 18870.166,E2 18870.166} C_VEL
LIN {X 0,Y 422.877,Z 428.188,A -85,B 0,C 180,E1 18868.696,E2 18868.696} C_VEL
LIN {X 0,Y 429.613,Z 437.06,A -85,B 0,C 180,E1 18866.963,E2 18866.963} C_VEL
LIN {X 0,Y 439.399,Z 450.555,A -85,B 0,C 180,E1 18864.651,E2 18864.651} C_VEL
LIN {X 0,Y 446.243,Z 460.889,A -85,B 0,C 180,E1 18863.144,E2 18863.144} C_VEL
LIN {X 0,Y 437.236,Z 671.812,A -85,B 0,C 180,E1 18859.217,E2 18859.217} C_VEL
LIN {X 0,Y 435.106,Z 717.726,A -85,B 0,C 180,E1 18858.334,E2 18858.334} C_VEL
LIN {X 0,Y 433.053,Z 740.23,A -85,B 0,C 180,E1 18857.698,E2 18857.698} C_VEL
LIN {X 0,Y 430.28,Z 763.581,A -85,B 0,C 180,E1 18856.801,E2 18856.801} C_VEL
LIN {X 0,Y 427.388,Z 782.963,A -85,B 0,C 180,E1 18855.847,E2 18855.847} C_VEL
LIN {X 0,Y 423.551,Z 805.056,A -85,B 0,C 180,E1 18854.51,E2 18854.51} C_VEL
LIN {X 0,Y 419.961,Z 823.067,A -85,B 0,C 180,E1 18853.189,E2 18853.189} C_VEL
LIN {X 0,Y 415.522,Z 843.376,A -85,B 0,C 180,E1 18851.425,E2 18851.425} C_VEL
LIN {X 0,Y 411.234,Z 861.413,A -85,B 0,C 180,E1 18849.564,E2 18849.564} C_VEL
LIN {X 0,Y 406.616,Z 879.968,A -85,B 0,C 180,E1 18847.305,E2 18847.305} C_VEL
LIN {X 0,Y 404.155,Z 889.548,A -85,B 0,C 180,E1 18845.986,E2 18845.986} C_VEL
LIN {X 0,Y 401.894,Z 895.061,A -85,B 0,C 180,E1 18845.26,E2 18845.26} C_VEL
LIN {X 0,Y 393.16,Z 908.838,A -85,B 0,C 180,E1 18843.554,E2 18843.554} C_VEL
LIN {X 0,Y 390.979,Z 913.685,A -85,B 0,C 180,E1 18842.748,E2 18842.748} C_VEL
LIN {X 0,Y 386.963,Z 928.588,A -85,B 0,C 180,E1 18839.738,E2 18839.738} C_VEL
LIN {X 0,Y 383.933,Z 940.371,A -85,B 0,C 180,E1 18836.941,E2 18836.941} C_VEL
LIN {X 0,Y 381.137,Z 952.118,A -85,B 0,C 180,E1 18833.661,E2 18833.661} C_VEL
LIN {X 0,Y 379.153,Z 961.56,A -85,B 0,C 180,E1 18830.529,E2 18830.529} C_VEL
LIN {X 0,Y 377.642,Z 970.083,A -85,B 0,C 180,E1 18827.088,E2 18827.088} C_VEL
LIN {X 0,Y 376.736,Z 976.822,A -85,B 0,C 180,E1 18823.744,E2 18823.744} C_VEL
LIN {X 0,Y 376.204,Z 981.928,A -85,B 0,C 180,E1 18820.41,E2 18820.41} C_VEL
LIN {X 0,Y 375.998,Z 985.271,A -85,B 0,C 180,E1 18817.486,E2 18817.486} C_VEL
LIN {X 0,Y 375.933,Z 987.849,A -85,B 0,C 180,E1 18813.964,E2 18813.964} C_VEL
LIN {X 0,Y 375.915,Z 988.764,A -85,B 0,C 180,E1 18811.066,E2 18811.066} C_VEL
LIN {X 0,Y 375.928,Z 988.625,A -85,B 0,C 180,E1 18807.866,E2 18807.866} C_VEL
LIN {X 0,Y 375.95,Z 986.971,A -85,B 0,C 180,E1 18804.506,E2 18804.506} C_VEL
LIN {X 0,Y 376.075,Z 984.278,A -85,B 0,C 180,E1 18801.438,E2 18801.438} C_VEL
LIN {X 0,Y 376.424,Z 979.514,A -85,B 0,C 180,E1 18797.819,E2 18797.819} C_VEL
LIN {X 0,Y 377.044,Z 974.201,A -85,B 0,C 180,E1 18794.781,E2 18794.781} C_VEL
LIN {X 0,Y 378.321,Z 966.056,A -85,B 0,C 180,E1 18791.112,E2 18791.112} C_VEL
LIN {X 0,Y 380.077,Z 957.093,A -85,B 0,C 180,E1 18787.82,E2 18787.82} C_VEL
LIN {X 0,Y 382.441,Z 946.501,A -85,B 0,C 180,E1 18784.614,E2 18784.614} C_VEL
LIN {X 0,Y 385.473,Z 934.448,A -85,B 0,C 180,E1 18781.496,E2 18781.496} C_VEL
LIN {X 0,Y 389.013,Z 920.889,A -85,B 0,C 180,E1 18778.553,E2 18778.553} C_VEL
LIN {X 0,Y 393.323,Z 905.196,A -85,B 0,C 180,E1 18775.647,E2 18775.647} C_VEL
LIN {X 0,Y 397.507,Z 889.911,A -85,B 0,C 180,E1 18773.231,E2 18773.231} C_VEL
LIN {X 0,Y 402.245,Z 872.249,A -85,B 0,C 180,E1 18770.854,E2 18770.854} C_VEL
LIN {X 0,Y 406.678,Z 855.135,A -85,B 0,C 180,E1 18768.882,E2 18768.882} C_VEL
LIN {X 0,Y 411.297,Z 835.804,A -85,B 0,C 180,E1 18766.999,E2 18766.999} C_VEL
LIN {X 0,Y 415.65,Z 816.226,A -85,B 0,C 180,E1 18765.385,E2 18765.385} C_VEL
LIN {X 0,Y 419.646,Z 795.624,A -85,B 0,C 180,E1 18763.989,E2 18763.989} C_VEL
LIN {X 0,Y 423.343,Z 774.133,A -85,B 0,C 180,E1 18762.789,E2 18762.789} C_VEL
LIN {X 0,Y 426.314,Z 752.7,A -85,B 0,C 180,E1 18761.853,E2 18761.853} C_VEL
LIN {X 0,Y 428.881,Z 729.516,A -85,B 0,C 180,E1 18761.077,E2 18761.077} C_VEL
LIN {X 0,Y 430.479,Z 707.862,A -85,B 0,C 180,E1 18760.562,E2 18760.562} C_VEL
LIN {X 0,Y 439.71,Z 500.411,A -85,B 0,C 180,E1 18756.669,E2 18756.669} C_VEL
LIN {X 0,Y 441.285,Z 464.645,A -85,B 0,C 180,E1 18755.98,E2 18755.98} C_VEL
LIN {X 0,Y 431.117,Z 449.906,A -85,B 0,C 180,E1 18753.623,E2 18753.623} C_VEL
LIN {X 0,Y 421.333,Z 436.544,A -85,B 0,C 180,E1 18751.114,E2 18751.114} C_VEL
LIN {X 0,Y 413.15,Z 426.101,A -85,B 0,C 180,E1 18748.79,E2 18748.79} C_VEL
LIN {X 0,Y 408.825,Z 420.707,A -85,B 0,C 180,E1 18747.453,E2 18747.453} C_VEL
LIN {X 0,Y 404.5,Z 415.386,A -85,B 0,C 180,E1 18746.024,E2 18746.024} C_VEL
LIN {X 0,Y 400.922,Z 411.244,A -85,B 0,C 180,E1 18744.77,E2 18744.77} C_VEL
LIN {X 0,Y 399.669,Z 409.566,A -85,B 0,C 180,E1 18744.301,E2 18744.301} C_VEL
LIN {X 0,Y 396.289,Z 406.046,A -85,B 0,C 180,E1 18743.022,E2 18743.022} C_VEL
LIN {X 0,Y 394.661,Z 403.576,A -85,B 0,C 180,E1 18742.335,E2 18742.335} C_VEL
LIN {X 0,Y 391.422,Z 400.748,A -85,B 0,C 180,E1 18740.994,E2 18740.994} C_VEL
LIN {X 0,Y 389.307,Z 397.332,A -85,B 0,C 180,E1 18739.974,E2 18739.974} C_VEL
LIN {X 0,Y 385.868,Z 394.835,A -85,B 0,C 180,E1 18738.351,E2 18738.351} C_VEL
LIN {X 0,Y 384.047,Z 391.674,A -85,B 0,C 180,E1 18737.305,E2 18737.305} C_VEL
LIN {X 0,Y 383.65,Z 390.708,A -85,B 0,C 180,E1 18737.05,E2 18737.05} C_VEL
LIN {X 0,Y 380.186,Z 388.861,A -85,B 0,C 180,E1 18735.092,E2 18735.092} C_VEL
LIN {X 0,Y 378.287,Z 386.282,A -85,B 0,C 180,E1 18733.762,E2 18733.762} C_VEL
LIN {X 0,Y 377.674,Z 383.998,A -85,B 0,C 180,E1 18733.161,E2 18733.161} C_VEL
LIN {X 0,Y 377.671,Z 383.991,A -85,B 0,C 180,E1 18729.11,E2 18729.11} C_VEL
LIN {X 0,Y 377.664,Z 383.989,A -85,B 0,C 180,E1 18725.165,E2 18725.165} C_VEL
LIN {X 0,Y 377.663,Z 383.987,A -85,B 0,C 180,E1 18721.062,E2 18721.062} C_VEL
LIN {X 0,Y 377.651,Z 383.99,A -85,B 0,C 180,E1 18716.965,E2 18716.965} C_VEL
LIN {X 0,Y 377.655,Z 383.995,A -85,B 0,C 180,E1 18712.852,E2 18712.852} C_VEL
LIN {X 0,Y 377.651,Z 384.008,A -85,B 0,C 180,E1 18708.702,E2 18708.702} C_VEL
LIN {X 0,Y 377.643,Z 384.198,A -85,B 0,C 180,E1 18707.306,E2 18707.306} C_VEL
LIN {X 0,Y 378.593,Z 386.869,A -85,B 0,C 180,E1 18706.484,E2 18706.484} C_VEL
LIN {X 0,Y 380.67,Z 389.345,A -85,B 0,C 180,E1 18705.084,E2 18705.084} C_VEL
LIN {X 0,Y 383.793,Z 390.953,A -85,B 0,C 180,E1 18703.348,E2 18703.348} C_VEL
LIN {X 0,Y 385.486,Z 394.361,A -85,B 0,C 180,E1 18702.334,E2 18702.334} C_VEL
LIN {X 0,Y 388.386,Z 396.865,A -85,B 0,C 180,E1 18700.917,E2 18700.917} C_VEL
LIN {X 0,Y 389.557,Z 397.612,A -85,B 0,C 180,E1 18700.392,E2 18700.392} C_VEL
LIN {X 0,Y 391.674,Z 401.129,A -85,B 0,C 180,E1 18699.373,E2 18699.373} C_VEL
LIN {X 0,Y 395.27,Z 404.294,A -85,B 0,C 180,E1 18697.898,E2 18697.898} C_VEL
LIN {X 0,Y 398.22,Z 408.361,A -85,B 0,C 180,E1 18696.706,E2 18696.706} C_VEL
LIN {X 0,Y 400.512,Z 410.54,A -85,B 0,C 180,E1 18695.871,E2 18695.871} C_VEL
LIN {X 0,Y 403.735,Z 414.735,A -85,B 0,C 180,E1 18694.71,E2 18694.71} C_VEL
LIN {X 0,Y 408.684,Z 421.194,A -85,B 0,C 180,E1 18693.05,E2 18693.05} C_VEL
LIN {X 0,Y 413.165,Z 427.306,A -85,B 0,C 180,E1 18691.646,E2 18691.646} C_VEL
LIN {X 0,Y 419.941,Z 436.637,A -85,B 0,C 180,E1 18689.685,E2 18689.685} C_VEL
LIN {X 0,Y 430.369,Z 451.983,A -85,B 0,C 180,E1 18686.95,E2 18686.95} C_VEL
LIN {X 0,Y 440.976,Z 469.035,A -85,B 0,C 180,E1 18684.439,E2 18684.439} C_VEL
LIN {X 0,Y 441.461,Z 470.275,A -85,B 0,C 180,E1 18684.318,E2 18684.318} C_VEL
LIN {X 0,Y 432.372,Z 674.865,A -85,B 0,C 180,E1 18680.481,E2 18680.481} C_VEL
LIN {X 0,Y 429.484,Z 738.014,A -85,B 0,C 180,E1 18679.274,E2 18679.274} C_VEL
LIN {X 0,Y 427.199,Z 761.243,A -85,B 0,C 180,E1 18678.645,E2 18678.645} C_VEL
LIN {X 0,Y 424.407,Z 783.257,A -85,B 0,C 180,E1 18677.844,E2 18677.844} C_VEL
LIN {X 0,Y 420.959,Z 804.881,A -85,B 0,C 180,E1 18676.811,E2 18676.811} C_VEL
LIN {X 0,Y 416.948,Z 826.844,A -85,B 0,C 180,E1 18675.507,E2 18675.507} C_VEL
LIN {X 0,Y 412.946,Z 846.128,A -85,B 0,C 180,E1 18674.111,E2 18674.111} C_VEL
LIN {X 0,Y 408.21,Z 867.11,A -85,B 0,C 180,E1 18672.294,E2 18672.294} C_VEL
LIN {X 0,Y 403.817,Z 885.175,A -85,B 0,C 180,E1 18670.44,E2 18670.44} C_VEL
LIN {X 0,Y 398.95,Z 904.204,A -85,B 0,C 180,E1 18668.141,E2 18668.141} C_VEL
LIN {X 0,Y 394.571,Z 921.213,A -85,B 0,C 180,E1 18665.735,E2 18665.735} C_VEL
LIN {X 0,Y 390.351,Z 937.278,A -85,B 0,C 180,E1 18663.061,E2 18663.061} C_VEL
LIN {X 0,Y 386.728,Z 951.791,A -85,B 0,C 180,E1 18660.272,E2 18660.272} C_VEL
LIN {X 0,Y 383.506,Z 965.117,A -85,B 0,C 180,E1 18657.248,E2 18657.248} C_VEL
LIN {X 0,Y 380.733,Z 977.881,A -85,B 0,C 180,E1 18653.853,E2 18653.853} C_VEL
LIN {X 0,Y 378.856,Z 987.826,A -85,B 0,C 180,E1 18650.708,E2 18650.708} C_VEL
LIN {X 0,Y 377.441,Z 996.88,A -85,B 0,C 180,E1 18647.257,E2 18647.257} C_VEL
LIN {X 0,Y 376.639,Z 1003.577,A -85,B 0,C 180,E1 18644.135,E2 18644.135} C_VEL
LIN {X 0,Y 376.145,Z 1009.52,A -85,B 0,C 180,E1 18640.568,E2 18640.568} C_VEL
LIN {X 0,Y 375.967,Z 1013.11,A -85,B 0,C 180,E1 18637.641,E2 18637.641} C_VEL
LIN {X 0,Y 375.922,Z 1015.854,A -85,B 0,C 180,E1 18634.271,E2 18634.271} C_VEL
LIN {X 0,Y 375.917,Z 1016.936,A -85,B 0,C 180,E1 18631.22,E2 18631.22} C_VEL
LIN {X 0,Y 375.922,Z 1016.866,A -85,B 0,C 180,E1 18628.324,E2 18628.324} C_VEL
LIN {X 0,Y 375.927,Z 1015.238,A -85,B 0,C 180,E1 18624.813,E2 18624.813} C_VEL
LIN {X 0,Y 376.016,Z 1012.452,A -85,B 0,C 180,E1 18621.746,E2 18621.746} C_VEL
LIN {X 0,Y 376.27,Z 1007.676,A -85,B 0,C 180,E1 18618.195,E2 18618.195} C_VEL
LIN {X 0,Y 376.801,Z 1002.021,A -85,B 0,C 180,E1 18615.087,E2 18615.087} C_VEL
LIN {X 0,Y 377.836,Z 994.234,A -85,B 0,C 180,E1 18611.647,E2 18611.647} C_VEL
LIN {X 0,Y 379.283,Z 985.484,A -85,B 0,C 180,E1 18608.508,E2 18608.508} C_VEL
LIN {X 0,Y 381.565,Z 973.998,A -85,B 0,C 180,E1 18605.047,E2 18605.047} C_VEL
LIN {X 0,Y 384.179,Z 962.292,A -85,B 0,C 180,E1 18602.069,E2 18602.069} C_VEL
LIN {X 0,Y 387.649,Z 947.903,A -85,B 0,C 180,E1 18598.95,E2 18598.95} C_VEL
LIN {X 0,Y 391.679,Z 932.338,A -85,B 0,C 180,E1 18596.061,E2 18596.061} C_VEL
LIN {X 0,Y 395.864,Z 916.065,A -85,B 0,C 180,E1 18593.506,E2 18593.506} C_VEL
LIN {X 0,Y 400.486,Z 898.369,A -85,B 0,C 180,E1 18591.111,E2 18591.111} C_VEL
LIN {X 0,Y 404.898,Z 880.721,A -85,B 0,C 180,E1 18589.081,E2 18589.081} C_VEL
LIN {X 0,Y 409.859,Z 859.859,A -85,B 0,C 180,E1 18587.041,E2 18587.041} C_VEL
LIN {X 0,Y 414.115,Z 840.643,A -85,B 0,C 180,E1 18585.468,E2 18585.468} C_VEL
LIN {X 0,Y 418.405,Z 819.15,A -85,B 0,C 180,E1 18584.011,E2 18584.011} C_VEL
LIN {X 0,Y 421.976,Z 798.933,A -85,B 0,C 180,E1 18582.885,E2 18582.885} C_VEL
LIN {X 0,Y 425.302,Z 776.447,A -85,B 0,C 180,E1 18581.893,E2 18581.893} C_VEL
LIN {X 0,Y 427.734,Z 756.457,A -85,B 0,C 180,E1 18581.211,E2 18581.211} C_VEL
LIN {X 0,Y 429.788,Z 732.312,A -85,B 0,C 180,E1 18580.611,E2 18580.611} C_VEL
LIN {X 0,Y 438.56,Z 532.701,A -85,B 0,C 180,E1 18576.86,E2 18576.86} C_VEL
LIN {X 0,Y 441.308,Z 469.665,A -85,B 0,C 180,E1 18575.65,E2 18575.65} C_VEL
LIN {X 0,Y 431.85,Z 454.47,A -85,B 0,C 180,E1 18573.438,E2 18573.438} C_VEL
LIN {X 0,Y 423.323,Z 441.671,A -85,B 0,C 180,E1 18571.263,E2 18571.263} C_VEL
LIN {X 0,Y 415.214,Z 429.964,A -85,B 0,C 180,E1 18568.987,E2 18568.987} C_VEL
LIN {X 0,Y 406.926,Z 418.798,A -85,B 0,C 180,E1 18566.406,E2 18566.406} C_VEL
LIN {X 0,Y 402.87,Z 413.853,A -85,B 0,C 180,E1 18565.033,E2 18565.033} C_VEL
LIN {X 0,Y 399.591,Z 409.521,A -85,B 0,C 180,E1 18563.835,E2 18563.835} C_VEL
LIN {X 0,Y 396.235,Z 405.951,A -85,B 0,C 180,E1 18562.564,E2 18562.564} C_VEL
LIN {X 0,Y 394.926,Z 403.733,A -85,B 0,C 180,E1 18562.005,E2 18562.005} C_VEL
LIN {X 0,Y 391.403,Z 400.792,A -85,B 0,C 180,E1 18560.563,E2 18560.563} C_VEL
LIN {X 0,Y 389.207,Z 397.252,A -85,B 0,C 180,E1 18559.509,E2 18559.509} C_VEL
LIN {X 0,Y 385.898,Z 394.883,A -85,B 0,C 180,E1 18557.958,E2 18557.958} C_VEL
LIN {X 0,Y 384.006,Z 391.566,A -85,B 0,C 180,E1 18556.877,E2 18556.877} C_VEL
LIN {X 0,Y 383.664,Z 390.734,A -85,B 0,C 180,E1 18556.658,E2 18556.658} C_VEL
LIN {X 0,Y 379.933,Z 388.708,A -85,B 0,C 180,E1 18554.556,E2 18554.556} C_VEL
LIN {X 0,Y 378.125,Z 385.873,A -85,B 0,C 180,E1 18553.261,E2 18553.261} C_VEL
LIN {X 0,Y 377.621,Z 383.994,A -85,B 0,C 180,E1 18552.773,E2 18552.773} C_VEL
LIN {X 0,Y 377.625,Z 383.994,A -85,B 0,C 180,E1 18548.833,E2 18548.833} C_VEL
LIN {X 0,Y 377.633,Z 383.995,A -85,B 0,C 180,E1 18544.86,E2 18544.86} C_VEL
LIN {X 0,Y 377.653,Z 383.996,A -85,B 0,C 180,E1 18540.91,E2 18540.91} C_VEL
LIN {X 0,Y 377.655,Z 384.004,A -85,B 0,C 180,E1 18536.812,E2 18536.812} C_VEL
LIN {X 0,Y 377.667,Z 384.004,A -85,B 0,C 180,E1 18532.699,E2 18532.699} C_VEL
LIN {X 0,Y 377.662,Z 383.994,A -85,B 0,C 180,E1 18528.547,E2 18528.547} C_VEL
LIN {X 0,Y 377.705,Z 384.231,A -85,B 0,C 180,E1 18526.568,E2 18526.568} C_VEL
LIN {X 0,Y 378.51,Z 386.781,A -85,B 0,C 180,E1 18525.857,E2 18525.857} C_VEL
LIN {X 0,Y 380.849,Z 389.413,A -85,B 0,C 180,E1 18524.311,E2 18524.311} C_VEL
LIN {X 0,Y 383.804,Z 391.004,A -85,B 0,C 180,E1 18522.684,E2 18522.684} C_VEL
LIN {X 0,Y 385.447,Z 394.32,A -85,B 0,C 180,E1 18521.707,E2 18521.707} C_VEL
LIN {X 0,Y 388.675,Z 397.032,A -85,B 0,C 180,E1 18520.149,E2 18520.149} C_VEL
LIN {X 0,Y 389.686,Z 397.801,A -85,B 0,C 180,E1 18519.694,E2 18519.694} C_VEL
LIN {X 0,Y 392.148,Z 401.638,A -85,B 0,C 180,E1 18518.538,E2 18518.538} C_VEL
LIN {X 0,Y 395.195,Z 404.22,A -85,B 0,C 180,E1 18517.304,E2 18517.304} C_VEL
LIN {X 0,Y 398.064,Z 408.216,A -85,B 0,C 180,E1 18516.146,E2 18516.146} C_VEL
LIN {X 0,Y 400.365,Z 410.352,A -85,B 0,C 180,E1 18515.311,E2 18515.311} C_VEL
LIN {X 0,Y 403.59,Z 414.584,A -85,B 0,C 180,E1 18514.149,E2 18514.149} C_VEL
LIN {X 0,Y 405.545,Z 416.657,A -85,B 0,C 180,E1 18513.496,E2 18513.496} C_VEL
LIN {X 0,Y 409.336,Z 421.195,A -85,B 0,C 180,E1 18512.269,E2 18512.269} C_VEL
LIN {X 0,Y 415.593,Z 429.32,A -85,B 0,C 180,E1 18510.369,E2 18510.369} C_VEL
LIN {X 0,Y 422.149,Z 437.59,A -85,B 0,C 180,E1 18508.556,E2 18508.556} C_VEL
LIN {X 0,Y 433.092,Z 452.743,A -85,B 0,C 180,E1 18505.795,E2 18505.795} C_VEL
LIN {X 0,Y 441.317,Z 464.97,A -85,B 0,C 180,E1 18503.903,E2 18503.903} C_VEL
LIN {X 0,Y 431.921,Z 675.221,A -85,B 0,C 180,E1 18499.963,E2 18499.963} C_VEL
LIN {X 0,Y 429.813,Z 718.206,A -85,B 0,C 180,E1 18499.127,E2 18499.127} C_VEL
LIN {X 0,Y 427.684,Z 740.676,A -85,B 0,C 180,E1 18498.488,E2 18498.488} C_VEL
LIN {X 0,Y 424.818,Z 763.893,A -85,B 0,C 180,E1 18497.592,E2 18497.592} C_VEL
LIN {X 0,Y 421.811,Z 783.275,A -85,B 0,C 180,E1 18496.633,E2 18496.633} C_VEL
LIN {X 0,Y 417.821,Z 805.366,A -85,B 0,C 180,E1 18495.287,E2 18495.287} C_VEL
LIN {X 0,Y 414.078,Z 823.377,A -85,B 0,C 180,E1 18493.958,E2 18493.958} C_VEL
LIN {X 0,Y 409.446,Z 843.687,A -85,B 0,C 180,E1 18492.18,E2 18492.18} C_VEL
LIN {X 0,Y 404.953,Z 861.725,A -85,B 0,C 180,E1 18490.302,E2 18490.302} C_VEL
LIN {X 0,Y 400.102,Z 880.281,A -85,B 0,C 180,E1 18488.019,E2 18488.019} C_VEL
LIN {X 0,Y 395.75,Z 896.388,A -85,B 0,C 180,E1 18485.7,E2 18485.7} C_VEL
LIN {X 0,Y 391.496,Z 911.763,A -85,B 0,C 180,E1 18483.102,E2 18483.102} C_VEL
LIN {X 0,Y 390.979,Z 913.685,A -85,B 0,C 180,E1 18482.748,E2 18482.748} C_VEL
LIN {X 0,Y 388.818,Z 918.569,A -85,B 0,C 180,E1 18481.912,E2 18481.912} C_VEL
LIN {X 0,Y 380.216,Z 930.608,A -85,B 0,C 180,E1 18479.881,E2 18479.881} C_VEL
LIN {X 0,Y 378.162,Z 934.959,A -85,B 0,C 180,E1 18478.963,E2 18478.963} C_VEL
LIN {X 0,Y 374.916,Z 947.076,A -85,B 0,C 180,E1 18475.763,E2 18475.763} C_VEL
LIN {X 0,Y 372.343,Z 957.844,A -85,B 0,C 180,E1 18472.412,E2 18472.412} C_VEL
LIN {X 0,Y 370.489,Z 966.736,A -85,B 0,C 180,E1 18469.057,E2 18469.057} C_VEL
LIN {X 0,Y 369.143,Z 974.684,A -85,B 0,C 180,E1 18465.364,E2 18465.364} C_VEL
LIN {X 0,Y 368.473,Z 980.035,A -85,B 0,C 180,E1 18462.217,E2 18462.217} C_VEL
LIN {X 0,Y 368.099,Z 984.645,A -85,B 0,C 180,E1 18458.59,E2 18458.59} C_VEL
LIN {X 0,Y 367.957,Z 987.317,A -85,B 0,C 180,E1 18455.456,E2 18455.456} C_VEL
LIN {X 0,Y 367.931,Z 988.934,A -85,B 0,C 180,E1 18452.024,E2 18452.024} C_VEL
LIN {X 0,Y 367.916,Z 989.077,A -85,B 0,C 180,E1 18448.91,E2 18448.91} C_VEL
LIN {X 0,Y 367.94,Z 988.123,A -85,B 0,C 180,E1 18445.792,E2 18445.792} C_VEL
LIN {X 0,Y 368.014,Z 985.663,A -85,B 0,C 180,E1 18442.35,E2 18442.35} C_VEL
LIN {X 0,Y 368.24,Z 982.346,A -85,B 0,C 180,E1 18439.361,E2 18439.361} C_VEL
LIN {X 0,Y 368.821,Z 977.157,A -85,B 0,C 180,E1 18435.879,E2 18435.879} C_VEL
LIN {X 0,Y 369.785,Z 970.584,A -85,B 0,C 180,E1 18432.536,E2 18432.536} C_VEL
LIN {X 0,Y 371.405,Z 962.113,A -85,B 0,C 180,E1 18429.022,E2 18429.022} C_VEL
